// TwinCAT 3 PLC project machine1
// ProgramVersion: 3.1.4026.23
// CompilerDefines: VISU_USEPROPERTYINFO
// libraries:
//   CmpBitmapPool, * (System)
//   Tc2_Standard, * (Beckhoff Automation GmbH)
//   Tc2_System, * (Beckhoff Automation GmbH)
//   Tc2_Utilities, * (Beckhoff Automation GmbH)
//   Tc3_IotBase, * (Beckhoff Automation GmbH)
//   VisuDialogs, * (System)
// project tree:
//   DUTs/ E_SeqState.TcDUT
//   / GlobalTextList.TcGTLO, ImagePool.TcIPO (not stored), PlcTask.TcTTO, VisualizationManager.TcVMO (not stored)
//   GVLs/ GVL_IO.TcGVL, GVL_Nav.TcGVL, GVL_Param.TcGVL, GVL_Process.TcGVL, GVL_Secrets.TcGVL (not stored)
//   POUs/ FB_EventLog.TcPOU, MAIN.TcPOU, PRG_FileLogger.TcPOU, PRG_Params.TcPOU, PRG_Process.TcPOU, PRG_Spray.TcPOU, PRG_StatsLogger.TcPOU, PRG_Telegram.TcPOU, SIM_Plant.TcPOU
//   VISUs/ visu_Nav.TcVIS, visu_Params.TcVIS, visu_Spray.TcVIS
// real-time tasks:
//   TASK PlcTask: cycle T#10ms, priority 20, ADS port 350
// I/O:
//   DEVICE Device 1 (EtherCAT), AmsNetId 192.168.1.120.2.1
//     Term 1 (EK1100) [EK1100 EtherCAT Coupler (2A E-Bus)]
//       Term 2 (EL1859) [EL1859 8Ch. Dig. Input 24V, 3ms, 8Ch. Dig. Output 24V, 0.5A]
//       Term 3 (EL3054) [EL3054 4Ch. Ana. Input 4-20mA]
//       Term 4 (EL9011) [EL9011 End Terminal]
// variable links:
//   machine1/machine1 Instance <-> Device 1 (EtherCAT)/Term 1 (EK1100)/Term 2 (EL1859)
//     PlcTask Outputs/GVL_IO.bAirValve <-> Channel 9/Output
//   machine1/machine1 Instance <-> Device 1 (EtherCAT)/Term 1 (EK1100)/Term 3 (EL3054)
//     PlcTask Inputs/GVL_IO.iSPXLevelRaw <-> AI Standard Channel 1/Value

CONFIGURATION machine1
    RESOURCE PLC ON TwinCAT3
        TASK PlcTask(INTERVAL := T#10ms, PRIORITY := 20);
        PROGRAM MAIN WITH PlcTask : MAIN;
    END_RESOURCE
END_CONFIGURATION

// ---- DUTs/E_SeqState.TcDUT

{attribute 'strict'}
{attribute 'to_string'}
TYPE E_SeqState :
(
    eIdle         := 0,    // S0 - outputs safe, circulation on; wait for the mother handshake
    eDewater      := 10,   // S1 - T1 dewater (suck slurry); move mold to spray height
    eSprayOpen    := 20,   // S2 - open Air+SPX, piston OPENING; watchdogs T2 (valve) & T3 (piston)
    eSprayClose   := 30,   // S3 - piston CLOSING; watchdog T4; spraying continues
    eCloseDewater := 40,   // S4 - close Air+SPX (watchdog T6); T5 dewater; then release mother
    eFault        := 100   // FAULT - safe, latched until reset
) INT;
END_TYPE

// ---- GVLs/GVL_IO.TcGVL
// Physical process I/O, named per the Alfa/Brazil spec.
// Moved out of MAIN's VAR_INPUT/VAR_OUTPUT because several programs now
// touch these signals (MAIN sequence, PRG_Process supervision, PRG_Spray
// HMI, SIM_Plant). A GVL is the standard shared home - same reason the
// machine parameters already live in GVL_Param.
//
// For real hardware: replace ';' with the AT %I*/%Q* mappings noted on
// each line and set SIM_Plant.bSimEnable := FALSE.
{attribute 'qualified_only'}
VAR_GLOBAL
    // ============ DIGITAL INPUTS (0-24 V) ============
    // ---- SPX-valve traffic-light feedback ----
    bSPXFullyOpen    : BOOL;   // SPX valve reported FULLY OPEN     // AT %I*
    bSPXFullyClose   : BOOL;   // SPX valve reported FULLY CLOSED   // AT %I*
    // ---- piston position sensors (from the mother machine) ----
    bPistonClosed    : BOOL;   // 'P-close' - piston at closed end  // AT %I*
    bPistonOpen      : BOOL;   // 'P-open'  - piston at open end    // AT %I*
    // ---- mother-machine handshake ----
    bSprayFeasible   : BOOL;   // mother in position & waiting: we may run   // AT %I*
    bMoldAtSprayHigh : BOOL;   // 'spray height' - mold reached spray pos    // AT %I*
    // ---- operator pushbuttons (OR-ed with the HMI buttons in MAIN) ----
    bAutoToggleHW    : BOOL;   // HW AUTO/STOP toggle               // AT %I*
    bResetHW         : BOOL;   // HW fault reset                    // AT %I*

    // ============ ANALOG INPUTS (4-20 mA, scaled to engineering units) ============
	iSPXLevelRaw  AT %I* : INT; 
    rSPXLevel        : REAL;   // SPX tank level  [%]               // AT %I* (scaled)
    rSPXPressure     : REAL;   // SPX pressure    [bar]             // AT %I* (scaled)
    rAirPressure     : REAL;   // Air pressure    [bar]             // AT %I* (scaled)
    rPumpHzFb        : REAL;   // gear-pump ACTUAL speed [Hz]       // AT %I* (scaled)
                               // VFD speed feedback - the MEASURED counterpart of
                               // the rPumpHz setpoint below. The mimic (pump circle
                               // + Hz readout) shows this, never the command, so a
                               // dead drive cannot look like a running one.

    // ============ DIGITAL OUTPUTS (0-24 V) ============
    bAirValve  AT %Q*      : BOOL;   // air valve solenoid                // AT %Q*
    bSPXValve        : BOOL;   // SPX valve - command OPEN          // AT %Q*
    bCircValve       : BOOL;   // circulation valve = NOT bSPXValve // AT %Q*
    bPistonOpenSol   : BOOL;   // piston OPEN  solenoid (or mother cmd)  // AT %Q*
    bPistonCloseSol  : BOOL;   // piston CLOSE solenoid (or mother cmd)  // AT %Q*
    bGoToCleaningPos : BOOL;   // command mother: move mold to spray height  // AT %Q*
    bSprayBusy       : BOOL;   // handshake to mother: we are running (mother waits)  // AT %Q*

    // ============ ANALOG OUTPUT (4-20 mA) ============
    rPumpHz          : REAL;   // gear-pump VFD speed setpoint [Hz] // AT %Q* (scaled)
END_VAR

// ---- GVLs/GVL_Nav.TcGVL
// Navigation state shared by the screen programs.
// Two screens now, per the spec.
{attribute 'qualified_only'}
VAR_GLOBAL
    nPage       : INT;                   // 0 = Spray System, 1 = Machine Parameters
    abNavActive : ARRAY[0..1] OF BOOL;   // highlight for the active nav button
END_VAR

// ---- GVLs/GVL_Param.TcGVL
// Machine parameters - persistent, writable from PRG_Params, read everywhere.
// Defaults match the "Machine Parameters" screen in the spec.
//   *** marks values the spec left open ("??"/"X"); tune on the machine. ***
{attribute 'qualified_only'}
VAR_GLOBAL PERSISTENT
    // ===== sequence timers (HMI "Machine Parameters" page) =====
    tDewaterTime       : TIME := T#4S;     // T1 - dewater / suck slurry            [operator]
    tSPXMaxOpenTime    : TIME := T#500MS;  // T2 - SPX valve must report OPEN  within this  [engineer]
    tSPXMaxCloseTime   : TIME := T#500MS;  // T6 - SPX valve must report CLOSE within this  [engineer]  (HMI groups T2&T6)
    tSprayOpenTime     : TIME := T#3S;     // T3 - piston OPEN  stroke watchdog (P-close->P-open) [engineer]
    tSprayCloseTime    : TIME := T#3S;     // T4 - piston CLOSE stroke watchdog (P-open->P-close) [engineer]  (HMI groups T3&T4)
    tSPXDewaterTime    : TIME := T#10S;    // T5 - dewater after closing            [operator]

    // ===== pressure / pump (HMI "Machine Parameters" page) =====
    rSPXPressureTarget : REAL := 1.7;      // SPX target pressure [bar]
    rPumpSpeedBase     : REAL := 15.0;     // gear-pump base speed [Hz] (P-control starts here)

    // ===== thresholds & gains (engineer; not on the operator page) =====
    rSPXPressTol       : REAL := 0.1;      // |avg-target| >= this  -> "bad SPX pressure" warning
    rPumpDeadband      : REAL := 0.02;     // P-control deadband [bar]
    rPumpKp            : REAL := 2.0;      // *** P-control gain [Hz per bar] - spec: "double the difference??" ***
    rPumpHzMin         : REAL := 5.0;      // *** pump speed clamp, low  [Hz] ***
    rPumpHzMax         : REAL := 50.0;     // *** pump speed clamp, high [Hz] ***
    rLevelHigh         : REAL := 95.0;     // SPX tank: warn above [%]
    rLevelLow          : REAL := 20.0;     // SPX tank: warn below [%]
    rLevelEmpty        : REAL := 5.0;      // SPX tank: below -> stop pump & block mother release [%]
    rCircPressTol      : REAL := 0.5;      // spray-avg vs circulation-avg > this -> "adjust" message

    // ===== logging =====
    // Directory for the event log file (PRG_FileLogger).
    //   ''  -> TwinCAT boot folder of the TARGET (portable default:
    //          Windows C:\TwinCAT\3.1\Boot\ , BSD/Linux /usr/local/etc/TwinCAT/3.1/Boot/)
    //   'C:\kayma\machine1'          -> Windows dev PC
    //   '/home/Administrator/logs'   -> Linux/BSD PLC (folder must exist & be writable
    //                                   by the TwinCAT runtime user!)
    // PERSISTENT: set once per machine, survives reboots. Takes effect on the
    // next logged event - no restart needed.
    sLogDir            : STRING(255) := '';

    // TRUE  -> every sequence state transition is logged as INFO
    //          (~4 extra lines per spray cycle; great for commissioning)
    // FALSE -> only cycle start/complete, faults, resets, warnings
    bLogStateChanges   : BOOL := TRUE;
	bStatsEnable   : BOOL := TRUE;   // master switch
    tStatsRun      : TIME := T#1S;   // sample period while cycle active
    tStatsIdle     : TIME := T#2M;   // keep-alive period idle/fault
    nStatsHourFrom : INT  := 0;      // daily window; From=To=0 -> 24h
    nStatsHourTo   : INT  := 0;      // e.g. 6 & 22 -> log 06:00-21:59
END_VAR

VAR_GLOBAL CONSTANT
    // ===== factory defaults (RESET button on the params page) =====
    // One authoritative home for the default machine parameters.
    // If you retune the machine, change the defaults HERE (they should
    // normally mirror the init values of the persistent block above).
    cDefDewaterTime    : TIME := T#4S;      // T1
    cDefValveMaxTime   : TIME := T#500MS;   // T2 & T6
    cDefSprayTime      : TIME := T#3S;      // T3 & T4
    cDefSPXDewaterTime : TIME := T#10S;     // T5
    cDefPressTarget    : REAL := 1.7;       // [bar]
    cDefPumpSpeed      : REAL := 15.0;      // [Hz]
END_VAR

// ---- GVLs/GVL_Process.TcGVL
// Derived process values + non-latching warnings.
//   - MAIN accumulates the SPX pressure averages during T3/T4.
//   - PRG_Process uses them for the end-of-cycle pump correction and
//     computes the level/circulation warnings.
//   - PRG_Spray shows them.
// (Sequence FAULTS are separate and latched - see MAIN.nErrorCode.)
{attribute 'qualified_only'}
VAR_GLOBAL
    // ---- SPX pressure averaging ----
    rSPXAvgT3      : REAL;   // "SPX Pressure average at T3"  (opening stroke)
    rSPXAvgT4      : REAL;   // "SPX Pressure average at T4"  (closing stroke)
    rSPXAvg        : REAL;   // "SPX Pressure average" = mean(T3, T4); drives pump P-control
    rSPXAvgCirc    : REAL;   // SPX pressure average during circulation (handshake down)

    // ---- warnings (non-latching; shown on the Spray screen) ----
    bWarnBadSPX    : BOOL;   // |spray avg - target| >= rSPXPressTol  ("bad SPX pressure")
    bWarnLevelHigh : BOOL;   // level > rLevelHigh
    bWarnLevelLow  : BOOL;   // level < rLevelLow
    bLevelEmpty    : BOOL;   // level < rLevelEmpty -> pump off + mother release blocked
    bWarnCircPress : BOOL;   // spray avg differs from circulation avg by > rCircPressTol ("adjust")
END_VAR

// ---- POUs/MAIN.TcPOU
PROGRAM MAIN
VAR_OUTPUT
    // ---- status (read by the HMI screens) ----
    eState        : E_SeqState := E_SeqState.eIdle;  // current sequence state
    nErrorCode    : INT;          // latched sequence fault (see constants)
    bAutoMode     : BOOL;         // TRUE = AUTO armed.  FALSE at boot = MANUAL
    bError        : BOOL;         // TRUE while in fault
    bReadyToStart : BOOL;         // TRUE while idle in manual (AUTO can be armed)
END_VAR

VAR
    // ---- edge detection ----
    rtAuto  : R_TRIG;   // AUTO/STOP toggle (HW OR HMI)
    rtReset : R_TRIG;   // fault reset      (HW OR HMI)

    // ---- timers (one per spec timer) ----
    tonDewater    : TON;   // T1 - dewater / suck slurry
    tonSPXOpen    : TON;   // T2 - SPX-valve-open watchdog
    tonSprayOpen  : TON;   // T3 - piston opening-stroke watchdog
    tonSprayClose : TON;   // T4 - piston closing-stroke watchdog
    tonSPXClose   : TON;   // T6 - SPX-valve-close watchdog
    tonDewaterCl  : TON;   // T5 - dewater after closing

    // ---- SPX pressure averaging accumulators ----
    rSumT3   : REAL;   nCntT3   : DINT;   // opening stroke
    rSumT4   : REAL;   nCntT4   : DINT;   // closing stroke
    rSumCirc : REAL;   nCntCirc : DINT;   // circulation (handshake down)
END_VAR

VAR CONSTANT
    // ---- latched fault codes ----
    nERR_NONE            : INT := 0;
    nERR_PISTON_NOT_HOME : INT := 10;   // start: piston not at P-close
    nERR_SPX_OPEN_STUCK  : INT := 20;   // T2: SPX valve never reported Fully Open
    nERR_SPX_CLOSE_STUCK : INT := 21;   // T6: SPX valve never reported Fully Close
    nERR_PISTON_OPEN_TO  : INT := 30;   // T3: piston did not reach P-open in time
    nERR_PISTON_CLOSE_TO : INT := 40;   // T4: piston did not reach P-close in time
	nERR_LEVEL_HIGH : INT := 50;   // SPX level above rLevelHigh (>95%)
	nERR_LEVEL_LOW  : INT := 51;   // SPX level below rLevelEmpty (<5%)
    nERR_UNKNOWN_STATE   : INT := 99;   // illegal eState

    // level fault auto-clear hysteresis [%]: the level must come back
    // this far INSIDE the band before the fault self-clears, so the
    // fault cannot chatter on/off right at the threshold.
    rLEVEL_CLEAR_HYST    : REAL := 2.0;
END_VAR

//==================================================================
// MAIN - spray sequence + scheduling   (aligned to the Alfa/Brazil spec)
//
// Flow (AUTO):  mother raises 'Spray feasible' -> we take control, move
// the mold to spray height, run ONE spray cycle (T1..T6), then lower
// 'busy' so the mother resumes. The cycle is handshake-gated, not free-
// running: each casting cycle the mother hands us control exactly once.
//==================================================================
SIM_Plant();    // drives GVL_IO inputs; bSimEnable is the sim/real master (HMI button)

// Scale EL3054 raw (0..32767 = 4..20 mA) -> SPX tank level [%].
// Only with REAL VALUES selected: while simulating, SIM_Plant ramps
// rSPXLevel and this must not overwrite it. Same single flag that
// gates every other input, so the level can never end up on a
// different source than the rest of the screen.
IF NOT SIM_Plant.bSimEnable THEN
    GVL_IO.rSPXLevel := INT_TO_REAL(GVL_IO.iSPXLevelRaw) * (100.0 / 32767.0);
END_IF

// Edge detectors (HW inputs OR-ed with the HMI buttons from PRG_Spray).
rtAuto (CLK := GVL_IO.bAutoToggleHW OR PRG_Spray.bCmdAuto);
rtReset(CLK := GVL_IO.bResetHW      OR PRG_Spray.bCmdReset);

// The circulation valve is ALWAYS the inverse of the SPX valve.
GVL_IO.bCircValve := NOT GVL_IO.bSPXValve;

// ---- AUTO / MANUAL toggle ----
//   press once  -> arm AUTO
//   AUTO -> MANUAL -> STOP NOW: abort to S0/idle on THIS scan. Because
//   this runs before the CASE, the eIdle branch below drops every
//   actuator the same scan - the running cycle stops immediately.
IF rtAuto.Q THEN
    IF bAutoMode THEN
        bAutoMode := FALSE;                 // AUTO -> MANUAL
        eState    := E_SeqState.eIdle;      // abort to S0 immediately (outputs drop in eIdle)
    ELSIF NOT bError THEN
        bAutoMode := TRUE;                  // arm AUTO
    END_IF
END_IF

CASE eState OF

    //--------------------------------------------------------------
    // S0 - IDLE / MANUAL   (circulation running, mother free)
    //--------------------------------------------------------------
    E_SeqState.eIdle:
        GVL_IO.bAirValve        := FALSE;
        GVL_IO.bSPXValve        := FALSE;     // -> circulation valve open
        GVL_IO.bPistonCloseSol  := TRUE;      // default: hold the piston closed
        GVL_IO.bPistonOpenSol   := FALSE;
        GVL_IO.bGoToCleaningPos := FALSE;
        GVL_IO.bSprayBusy       := FALSE;     // mother is free to move
        bError        := FALSE;
        bReadyToStart := NOT bAutoMode;
        nErrorCode    := nERR_NONE;

        // reset all timers + stroke accumulators (clean start next cycle)
        tonDewater(IN := FALSE);   tonSPXOpen(IN := FALSE);   tonSprayOpen(IN := FALSE);
        tonSprayClose(IN := FALSE); tonSPXClose(IN := FALSE); tonDewaterCl(IN := FALSE);
        rSumT3 := 0; nCntT3 := 0; rSumT4 := 0; nCntT4 := 0;

        // average SPX pressure during circulation (handshake down)
        rSumCirc := rSumCirc + GVL_IO.rSPXPressure;
        nCntCirc := nCntCirc + 1;
        IF nCntCirc > 0 THEN
            GVL_Process.rSPXAvgCirc := rSumCirc / DINT_TO_REAL(nCntCirc);
        END_IF

        IF bAutoMode THEN
            // Start a cycle only when the mother hands control over
            // (bSprayFeasible), the piston is home, and the tank isn't empty.
            IF GVL_IO.bSprayFeasible AND GVL_IO.bPistonClosed AND NOT GVL_Process.bLevelEmpty THEN
                GVL_IO.bSprayBusy       := TRUE;   // tell the mother we are running
                GVL_IO.bGoToCleaningPos := TRUE;   // ask the mother to move the mold up
                GVL_Process.bWarnBadSPX := FALSE;  // fresh cycle
                rSumCirc := 0; nCntCirc := 0;      // restart circulation average
                bReadyToStart := FALSE;
                eState := E_SeqState.eDewater;
            END_IF
        ELSIF PRG_Spray.bManualActive THEN
            // MANUAL: operator drives the actuators directly.
            GVL_IO.bAirValve       := PRG_Spray.bManAirValve;
            GVL_IO.bSPXValve       := PRG_Spray.bManSPXValve;
            GVL_IO.bPistonOpenSol  := PRG_Spray.bManPistonOpen;
            GVL_IO.bPistonCloseSol := PRG_Spray.bManPistonClose;
        END_IF

    //--------------------------------------------------------------
    // S1 - DEWATER (T1)   + position the mold to spray height
    //--------------------------------------------------------------
    E_SeqState.eDewater:
        GVL_IO.bAirValve       := FALSE;
        GVL_IO.bSPXValve       := FALSE;
        GVL_IO.bPistonCloseSol := TRUE;       // keep piston closed
        GVL_IO.bPistonOpenSol  := FALSE;

        // keep asking until the mold reports it is at spray height
        GVL_IO.bGoToCleaningPos := NOT GVL_IO.bMoldAtSprayHigh;

        tonDewater(IN := TRUE, PT := GVL_Param.tDewaterTime);

        // advance once T1 elapsed AND the mold is in position
        IF tonDewater.Q AND GVL_IO.bMoldAtSprayHigh THEN
            eState := E_SeqState.eSprayOpen;
        END_IF

    //--------------------------------------------------------------
    // S2 - SPRAY, OPENING   (open valves; piston travels P-close->P-open)
    //   T2 watchdog: SPX valve must reach Fully Open.
    //   T3 watchdog: piston must complete the opening stroke.
    //   Average SPX pressure over the stroke -> "...average at T3".
    //--------------------------------------------------------------
    E_SeqState.eSprayOpen:
        GVL_IO.bAirValve       := TRUE;
        GVL_IO.bSPXValve       := TRUE;       // -> circulation valve closes
        GVL_IO.bPistonOpenSol  := TRUE;       // drive piston OPEN
        GVL_IO.bPistonCloseSol := FALSE;

        // T2 - SPX-valve-open confirmation watchdog (runs until Fully Open)
        tonSPXOpen(IN := NOT GVL_IO.bSPXFullyOpen, PT := GVL_Param.tSPXMaxOpenTime);
        IF tonSPXOpen.Q THEN
            nErrorCode := nERR_SPX_OPEN_STUCK;
            eState     := E_SeqState.eFault;
        END_IF

        // T3 - opening-stroke watchdog (starts once the piston leaves P-close)
        tonSprayOpen(IN := NOT GVL_IO.bPistonClosed, PT := GVL_Param.tSprayOpenTime);
        IF tonSprayOpen.Q AND NOT GVL_IO.bPistonOpen THEN
            nErrorCode := nERR_PISTON_OPEN_TO;
            eState     := E_SeqState.eFault;
        END_IF

        // running SPX pressure average over the opening stroke
        rSumT3 := rSumT3 + GVL_IO.rSPXPressure;
        nCntT3 := nCntT3 + 1;

        // stroke finished -> store average, check pressure, go to closing
        IF GVL_IO.bPistonOpen THEN
            IF nCntT3 > 0 THEN
                GVL_Process.rSPXAvgT3 := rSumT3 / DINT_TO_REAL(nCntT3);
            END_IF
            IF ABS(GVL_Process.rSPXAvgT3 - GVL_Param.rSPXPressureTarget) >= GVL_Param.rSPXPressTol THEN
                GVL_Process.bWarnBadSPX := TRUE;
            END_IF
            eState := E_SeqState.eSprayClose;
        END_IF

    //--------------------------------------------------------------
    // S3 - SPRAY, CLOSING   (piston travels P-open->P-close)
    //   T4 watchdog: piston must complete the closing stroke.
    //   Average SPX pressure over the stroke -> "...average at T4".
    //--------------------------------------------------------------
    E_SeqState.eSprayClose:
        GVL_IO.bAirValve       := TRUE;
        GVL_IO.bSPXValve       := TRUE;
        GVL_IO.bPistonOpenSol  := FALSE;
        GVL_IO.bPistonCloseSol := TRUE;       // drive piston CLOSE

        // T4 - closing-stroke watchdog (starts once the piston leaves P-open)
        tonSprayClose(IN := NOT GVL_IO.bPistonOpen, PT := GVL_Param.tSprayCloseTime);
        IF tonSprayClose.Q AND NOT GVL_IO.bPistonClosed THEN
            nErrorCode := nERR_PISTON_CLOSE_TO;
            eState     := E_SeqState.eFault;
        END_IF

        rSumT4 := rSumT4 + GVL_IO.rSPXPressure;
        nCntT4 := nCntT4 + 1;

        IF GVL_IO.bPistonClosed THEN
            IF nCntT4 > 0 THEN
                GVL_Process.rSPXAvgT4 := rSumT4 / DINT_TO_REAL(nCntT4);
            END_IF
            IF ABS(GVL_Process.rSPXAvgT4 - GVL_Param.rSPXPressureTarget) >= GVL_Param.rSPXPressTol THEN
                GVL_Process.bWarnBadSPX := TRUE;
            END_IF
            eState := E_SeqState.eCloseDewater;
        END_IF

    //--------------------------------------------------------------
    // S4 - CLOSE + DEWATER   (T6 valve-close watchdog + T5 dewater)
    //   On T5 end: lower 'busy' -> the mother resumes.
    //--------------------------------------------------------------
    E_SeqState.eCloseDewater:
        GVL_IO.bAirValve       := FALSE;
        GVL_IO.bSPXValve       := FALSE;      // -> circulation valve opens again
        GVL_IO.bPistonOpenSol  := FALSE;
        GVL_IO.bPistonCloseSol := TRUE;       // hold piston closed

        // T6 - SPX-valve-close confirmation watchdog (runs until Fully Close)
        tonSPXClose(IN := NOT GVL_IO.bSPXFullyClose, PT := GVL_Param.tSPXMaxCloseTime);
        IF tonSPXClose.Q THEN
            nErrorCode := nERR_SPX_CLOSE_STUCK;
            eState     := E_SeqState.eFault;
        END_IF

        // T5 - dewater
        tonDewaterCl(IN := TRUE, PT := GVL_Param.tSPXDewaterTime);
        IF tonDewaterCl.Q THEN
            // tank-empty lockout: do NOT release the mother while empty
            IF NOT GVL_Process.bLevelEmpty THEN
                GVL_IO.bSprayBusy := FALSE;          // lower the flag -> mother resumes
                eState            := E_SeqState.eIdle;
            END_IF
        END_IF

    //--------------------------------------------------------------
    // FAULT - latched until reset.
    //   The actuators are forced safe by the SAFE-STATE OVERLAY right
    //   after this CASE, so a fault raised mid-cycle drops every output
    //   on the SAME scan (the spray states energise their outputs at the
    //   top of their branch, then test for faults).
    //--------------------------------------------------------------
    E_SeqState.eFault:
        // LEVEL faults (50/51) self-clear as soon as the operator brings
        // the tank back into band (refill after "low", drain after "high"),
        // with hysteresis so the fault can't chatter at the threshold.
        // Every other fault stays latched until Reset.
        // NOTE: the safe-state overlay already dropped AUTO -> MANUAL, so
        // after the auto-clear the machine sits safely in Idle/MANUAL and
        // the operator re-arms AUTO deliberately.
        IF rtReset.Q
        OR (nErrorCode = nERR_LEVEL_LOW  AND GVL_IO.rSPXLevel >= GVL_Param.rLevelEmpty + rLEVEL_CLEAR_HYST)
        OR (nErrorCode = nERR_LEVEL_HIGH AND GVL_IO.rSPXLevel <= GVL_Param.rLevelHigh  - rLEVEL_CLEAR_HYST) THEN
            bError     := FALSE;
            nErrorCode := nERR_NONE;
            eState     := E_SeqState.eIdle;
        END_IF

ELSE
    nErrorCode := nERR_UNKNOWN_STATE;
    eState     := E_SeqState.eFault;
END_CASE

//==================================================================
// SPX LEVEL FAULT - out-of-band level raises a latched fault,
//   but ONLY while AUTO is armed or a spray cycle is running.
//   >95% = overfill,  <5% = dry/disconnected.
//   In MANUAL + idle (operator draining / refilling / cleaning) NO
//   fault is raised - the machine is still protected by:
//     - the non-latching warnings on the Spray screen (PRG_Process)
//     - the tank-empty pump lockout in PRG_Process (pump -> 0 Hz)
//     - the AUTO start gate in eIdle (NOT bLevelEmpty)
//   The fault self-clears in eFault once the level is back in band
//   (see the eFault branch above); Reset also still works.
//==================================================================
IF eState <> E_SeqState.eFault AND (bAutoMode OR eState <> E_SeqState.eIdle) THEN
    IF GVL_IO.rSPXLevel > GVL_Param.rLevelHigh THEN
        nErrorCode := nERR_LEVEL_HIGH;
        eState     := E_SeqState.eFault;
    ELSIF GVL_IO.rSPXLevel < GVL_Param.rLevelEmpty THEN
        nErrorCode := nERR_LEVEL_LOW;
        eState     := E_SeqState.eFault;
    END_IF
END_IF

//==================================================================
// SAFE-STATE OVERLAY - runs every scan, right after the sequencer.
//   A fault must stop the process RIGHT AWAY. The spray states set
//   their outputs TRUE at the top of the branch and only then test for
//   faults, so without this the actuators would drop one scan late. On
//   the scan a fault is raised, eState is already eFault here, so every
//   output drops in the same scan and AUTO is dropped to MANUAL.
//   (The AUTO->MANUAL abort lands in eIdle above, which is safe the
//    same scan, so it needs no overlay.)
//==================================================================
IF eState = E_SeqState.eFault THEN
    GVL_IO.bAirValve        := FALSE;
    GVL_IO.bSPXValve        := FALSE;
    GVL_IO.bPistonOpenSol   := FALSE;
    GVL_IO.bPistonCloseSol  := TRUE;     // hold the piston closed
    GVL_IO.bGoToCleaningPos := FALSE;
    GVL_IO.bSprayBusy       := FALSE;    // hand control back to the mother
    bError        := TRUE;
    bReadyToStart := FALSE;
    bAutoMode     := FALSE;              // a fault always drops AUTO -> MANUAL
END_IF

//==================================================================
// Supervision + screen programs (all run every scan)
//==================================================================
PRG_Process();   // level monitoring, pump P-control, circulation check
PRG_Spray();     // Spray System screen      (page 0)
PRG_Params();    // Machine Parameters screen (page 1)
PRG_FileLogger(); // Logger for the machine
PRG_Telegram();  // Telegram fault notifier (TF6760)

END_PROGRAM

// ---- POUs/SIM_Plant.TcPOU
PROGRAM SIM_Plant
//==================================================================
// PLANT SIMULATOR - drives the GVL_IO *inputs* from the GVL_IO outputs
// so the aligned sequence can run without hardware. Stroke/valve times
// are set INSIDE the watchdog limits (T2/T3/T4/T6) so a clean demo
// never faults. Set bSimEnable := FALSE for real I/O.
//
// bSimEnable is the ONE switch: it is what the 'SIM VALUES / REAL
// VALUES' button on the spray screen toggles, and it covers every
// process input at once (level, pressures, pump speed feedback, valve
// traffic-light, piston sensors, mold-at-height, mother handshake).
// On the falling
// edge the simulated values are dropped rather than left latched -
// see the release block at the top of the implementation.
//==================================================================
VAR
    bSimEnable       : BOOL := TRUE;     // master enable (HMI: 'SIM VALUES' button)
    bSimAutoStart    : BOOL := FALSE;    // TRUE = kick the machine into AUTO once (demo).
                                         // Default FALSE: boots in MANUAL, as specified.
	ftSimOff        : F_TRIG;         // SIM -> REAL edge (release the sim values)
    fSimLevel       : REAL := 20.0;   // simulated level [%]
    fSimRate        : REAL := 5.0;    // rate of change [% per second]
    bSimUp          : BOOL := TRUE;   // TRUE = filling, FALSE = draining
	bAutoKicked 	: BOOL;
    tLast           : TIME;
    fDt             : REAL;

    // ---- simulated mechanical times (must stay < the matching watchdog) ----
    tSimPistonStroke : TIME := T#2S;     // piston travel  (< T3 / T4 = 3 s)
    tSimValveStroke  : TIME := T#300MS;  // SPX valve open/close (< T2 / T6 = 0.5 s)
    tSimMoldMove     : TIME := T#1S;     // mother moves mold to spray height (< T1 = 4 s)
    tSimStartGap     : TIME := T#2S;     // settle time before the demo auto-kick

    // ---- simulated VFD speed feedback ----
    rSimPumpLag      : REAL := 0.15;  // per-scan approach factor -> spin-up/down
    rSimPumpZero     : REAL := 0.5;   // [Hz] snap the lag tail to 0 below this.
                                      // Keep at/below PRG_Spray.rPUMP_RUN_MIN, the
                                      // threshold the mimic calls 'stopped'.

    // ---- timers ----
    tonPOpen   : TON;
    tonPClose  : TON;
    tonSPXO    : TON;
    tonSPXC    : TON;
    tonMold    : TON;
    tonStart   : TON;
    rtStartGap : R_TRIG;
    
END_VAR

//------------------------------------------------------------------
// Simulation off -> leave every input to the real I/O.
//   On the SIM -> REAL edge the values this program was writing are
//   cleared. Without that they stay latched at their last simulated
//   figure and keep reading like live measurements - the piston lamps
//   stay green, SPX still shows 1.72 bar - which is exactly the trap
//   the sim/real button exists to prevent. Zeroed inputs make an
//   unmapped or dead channel obvious immediately (and, in AUTO, the
//   existing watchdogs fault the cycle instead of running blind).
//------------------------------------------------------------------
ftSimOff(CLK := bSimEnable);

IF NOT bSimEnable THEN
    IF ftSimOff.Q THEN
        GVL_IO.rSPXPressure     := 0.0;
        GVL_IO.rAirPressure     := 0.0;
        GVL_IO.rPumpHzFb        := 0.0;
        GVL_IO.bSPXFullyOpen    := FALSE;
        GVL_IO.bSPXFullyClose   := FALSE;
        GVL_IO.bPistonOpen      := FALSE;
        GVL_IO.bPistonClosed    := FALSE;
        GVL_IO.bMoldAtSprayHigh := FALSE;
        GVL_IO.bSprayFeasible   := FALSE;
        GVL_IO.bAutoToggleHW    := FALSE;
        // rSPXLevel is not cleared here: MAIN scales it from the real
        // iSPXLevelRaw channel every scan as soon as sim is off.
    END_IF
    RETURN;
END_IF

//------------------------------------------------------------------
// Mother handshake: mother is always ready in the demo, so each time
// the cycle returns to idle it hands control over again (cycles loop).
//------------------------------------------------------------------
GVL_IO.bSprayFeasible := TRUE;

//------------------------------------------------------------------
// Piston position sensors (P-close / P-open) follow the solenoids.
//   leaving an end clears that end immediately; reaching the far end
//   takes tSimPistonStroke.
//------------------------------------------------------------------
tonPOpen (IN := GVL_IO.bPistonOpenSol,  PT := tSimPistonStroke);
tonPClose(IN := GVL_IO.bPistonCloseSol, PT := tSimPistonStroke);

IF GVL_IO.bPistonOpenSol THEN
    GVL_IO.bPistonClosed := FALSE;
    GVL_IO.bPistonOpen   := tonPOpen.Q;
ELSIF GVL_IO.bPistonCloseSol THEN
    GVL_IO.bPistonOpen   := FALSE;
    GVL_IO.bPistonClosed := tonPClose.Q;
END_IF

//------------------------------------------------------------------
// SPX valve traffic-light follows the SPX valve command.
//------------------------------------------------------------------
tonSPXO(IN := GVL_IO.bSPXValve,     PT := tSimValveStroke);
tonSPXC(IN := NOT GVL_IO.bSPXValve, PT := tSimValveStroke);

IF GVL_IO.bSPXValve THEN
    GVL_IO.bSPXFullyClose := FALSE;
    GVL_IO.bSPXFullyOpen  := tonSPXO.Q;
ELSE
    GVL_IO.bSPXFullyOpen  := FALSE;
    GVL_IO.bSPXFullyClose := tonSPXC.Q;
END_IF

//------------------------------------------------------------------
// Mold reaches spray height shortly after we take control (busy).
//------------------------------------------------------------------
tonMold(IN := GVL_IO.bSprayBusy, PT := tSimMoldMove);
GVL_IO.bMoldAtSprayHigh := tonMold.Q;

//------------------------------------------------------------------
// Analog inputs.  Level mid-range (no level warnings); SPX pressure
// eases toward ~1.72 bar while spraying (within tolerance of 1.70).
//------------------------------------------------------------------

IF GVL_IO.bSPXValve THEN
    GVL_IO.rSPXPressure := GVL_IO.rSPXPressure + (1.72 - GVL_IO.rSPXPressure) * 0.3;
ELSE
    GVL_IO.rSPXPressure := GVL_IO.rSPXPressure + (1.50 - GVL_IO.rSPXPressure) * 0.1;
END_IF

IF GVL_IO.bAirValve THEN
    GVL_IO.rAirPressure := GVL_IO.rAirPressure + (28.0 - GVL_IO.rAirPressure) * 0.3;
ELSE
    GVL_IO.rAirPressure := GVL_IO.rAirPressure + (5.0 - GVL_IO.rAirPressure) * 0.1;
END_IF

//------------------------------------------------------------------
// Gear-pump speed feedback: first-order lag toward the VFD setpoint,
// i.e. spin-up and spin-down instead of an instant jump. The setpoint
// read here is the one written LAST scan (PRG_Process / PRG_Spray both
// run after this program), which is the right way round - a real drive
// reports where it has got to, not where it was just told to go.
// Snapped to exactly 0 below the run threshold: the lag is asymptotic,
// and a stopped pump must read zero rather than leave a tail that
// keeps the mimic circle green forever.
//------------------------------------------------------------------
GVL_IO.rPumpHzFb := GVL_IO.rPumpHzFb + (GVL_IO.rPumpHz - GVL_IO.rPumpHzFb) * rSimPumpLag;
IF GVL_IO.rPumpHz <= 0.0 AND GVL_IO.rPumpHzFb < rSimPumpZero THEN
    GVL_IO.rPumpHzFb := 0.0;
END_IF

//------------------------------------------------------------------
// Demo kick-off: pulse the AUTO toggle ONCE after boot (if enabled).
// Cycles then loop on their own (machine stays armed in AUTO), so we
// must NOT pulse again - a second pulse would disarm AUTO.
//------------------------------------------------------------------
tonStart(IN := bSimAutoStart AND NOT bAutoKicked AND (MAIN.eState = E_SeqState.eIdle),
         PT := tSimStartGap);
rtStartGap(CLK := tonStart.Q);
GVL_IO.bAutoToggleHW := rtStartGap.Q;
IF rtStartGap.Q THEN
    bAutoKicked := TRUE;
END_IF

fDt   := TIME_TO_REAL(TIME() - tLast) / 1000.0;
tLast := TIME();
fDt   := LIMIT(0.0, fDt, 0.1);   // guard against the first-cycle jump

// Level ramp - unconditional while simulating, like every other value
// this program drives. (There used to be a bSimLevelActive sub-flag
// that could hold the level on the real channel while the rest of the
// screen was simulated; with bSimEnable on the HMI it was a second,
// unreachable switch that silently froze the level. One switch only.)
IF bSimUp THEN
    fSimLevel := fSimLevel + fSimRate * fDt;
    IF fSimLevel >= 90.0 THEN
        fSimLevel := 90.0;
        bSimUp    := FALSE;      // top reached -> drain
    END_IF
ELSE
    fSimLevel := fSimLevel - fSimRate * fDt;
    IF fSimLevel <= 21.0 THEN
        fSimLevel := 21.0;
        bSimUp    := TRUE;       // bottom reached -> fill
    END_IF
END_IF
GVL_IO.rSPXLevel := fSimLevel;

END_PROGRAM

// ---- POUs/PRG_Spray.TcPOU
PROGRAM PRG_Spray
//==================================================================
// SPRAY SYSTEM SCREEN  (page 0)
//   The mimic view from the spec (slide 12). Merges the three old
//   spray programs (process view + manual + live readouts) into one
//   schematic screen:
//     - valve states by colour: green = open, grey = closed,
//       red = in transit (SPX by traffic-light, circulation = inverse,
//       air by command)
//     - piston lamps (green at a known end), mold-at-height lamp,
//       spray marks, pump Hz, SPX level, SPX/Air pressures
//     - manual buttons (live only in manual); mode colour
//       yellow = manual, green = auto
//     - CLEAN MODE (manual only): drain tank -> close drain / add
//       water prompts -> refill to 20% -> 20 s delay -> auto-open
//       the SPX valve to flush the pipes (section 6b)
//   The sequence engine stays in MAIN; this program is the HMI face.
//==================================================================
VAR_OUTPUT
    // ---- operator commands consumed by MAIN ----
    bCmdAuto  : BOOL;    // AUTO/MANUAL toggle button (tap = pulse)
    bCmdReset : BOOL;    // "Reset fault" button

    // ---- manual mode (consumed by MAIN while idle) ----
    bManualActive   : BOOL;   // TRUE = manual commands drive the outputs
    bManAirValve    : BOOL;   // manual: air valve        (HMI toggle)
    bManSPXValve    : BOOL;   // manual: SPX valve         (HMI toggle)
    bManPistonOpen  : BOOL;   // manual: piston OPEN  sol. (HMI toggle)
    bManPistonClose : BOOL;   // manual: piston CLOSE sol. (HMI toggle)
    rManPumpHz      : REAL := 15.0;   // manual/clean pump speed [Hz] - mirrors GVL_Param.rPumpSpeedBase every scan

    // ---- clean mode (read by MAIN) ----
    bCleanActive    : BOOL;   // TRUE = clean sequence running: MAIN skips the
                              // level-LOW fault and refuses to arm AUTO
    bPostCleanEmpty : BOOL;   // TRUE = clean ended with a dry tank: keep the
                              // level-LOW fault suppressed until refilled >5%
END_VAR

VAR
	
 	// ---- readout text colours (AARRGGBB) ----
    //   black = normal, amber = warning, red = lockout. Driven from the flags
    //   PRG_Process/MAIN already evaluate, so the colour on screen can never
    //   disagree with the fault code or the log file.
    cSPXPress   : DWORD;   // SPX pressure field. Amber while GVL_Process.bWarnBadSPX,
                           // i.e. the last cycle's T3/T4 average sat further than
                           // rSPXPressTol from rSPXPressureTarget. Latched per cycle,
                           // so it describes the last spray, not the live number.
    cLevel      : DWORD;   // SPX level field. Amber below rLevelLow or above
                           // rLevelHigh, red below rLevelEmpty (bLevelEmpty, which
                           // also stops the pump and blocks the mother release).
    // ---- mimic colours (AARRGGBB) ----
    cAirValve   : DWORD;
    cSPXValve   : DWORD;
    cCircValve  : DWORD;
    cPistonOpen : DWORD;
    cPistonClose: DWORD;
    cModeColor  : DWORD;

    // ---- lamps / flags ----
    bMoldLamp   : BOOL;   // mold at spray height
    bSprayMarks : BOOL;   // spray marks visible
    bFault      : BOOL;

    // ---- text ----
    sStateText  : STRING;
    sModeText   : STRING;
    sErrorText  : STRING;
    sWarnText   : STRING;

    // ---- live readouts mirrored for the HMI ----
    rPumpHz      : REAL;
    rSPXLevel    : REAL;
    rSPXPressure : REAL;
    rAirPressure : REAL;

    // ---- clean mode: HMI buttons (Toggle inputs; consumed in section 7) ----
    bBtnClean      : BOOL;   // 'CLEAN MODE' / 'STOP CLEAN' button
    bBtnStartClean : BOOL;   // 'Start Clean' button
    bBtnCloseDrain : BOOL;   // 'Close Drain' acknowledge button
    bBtnAddWater   : BOOL;   // 'Add Water'  acknowledge button

    // ---- clean mode: state + HMI feedback ----
    nCleanStep     : INT;    // nCLEAN_* constants below
    bDrainAck      : BOOL;   // operator confirmed the drain is closed
    bWaterAck      : BOOL;   // operator confirmed water is being added
    bDrainFlash    : BOOL;   // bind to 'Close Drain' toggle-colour -> flashes
    bWaterFlash    : BOOL;   // bind to 'Add Water'  toggle-colour -> flashes
    sCleanBtnText  : STRING := 'CLEAN MODE';  // 'CLEAN MODE' <-> 'STOP CLEAN'
    sCleanStatus   : STRING; // one-line operator guidance + countdown
    nFlushSecsLeft : INT;    // countdown [s] before the SPX valve auto-opens

    tonFlush       : TON;    // delay before the flush (tFLUSH_DELAY)
    tonBlink       : TON;    // 0.5 s blink generator for the flashing buttons
    bBlinkPhase    : BOOL;
    bCleanPrev     : BOOL;   // clean-active on the previous scan (exit edge)

    i : INT;
	
	 // ---- water animation (spray strokes + clean flush) ----
    bWaterFlow : BOOL;                   // TRUE = stream visible
    abDrop     : ARRAY[0..3] OF BOOL;    // one flag per droplet, top -> bottom
    nDropIdx   : INT;                    // chaser position
    tonDrop    : TON;
    j          : INT;
END_VAR

VAR CONSTANT
    cGREEN  : DWORD := 16#FF46A758;   // open / auto / OK
    cGREY   : DWORD := 16#FF8A8F98;   // closed
    cRED    : DWORD := 16#FFE5484D;   // in transit / fault
    cYELLOW : DWORD := 16#FFF2C94C;   // manual
	cBLACK  : DWORD := 16#FF000000;

    // ---- clean-mode steps ----
    nCLEAN_OFF       : INT := 0;   // clean mode not active
    nCLEAN_READY     : INT := 1;   // entered clean; waiting for Start Clean
    nCLEAN_DRAIN     : INT := 2;   // pump runs until the tank reads ~0 %
    nCLEAN_ACK       : INT := 3;   // pump off; Close Drain + Add Water flash
    nCLEAN_REFILL    : INT := 4;   // acks done; wait level >= 20 % + Start Clean
    nCLEAN_FLUSHWAIT : INT := 5;   // 20 s countdown, then SPX auto-opens
    nCLEAN_FLUSH     : INT := 6;   // SPX open, pump flushes the pipes

    rCLEAN_EMPTY : REAL := 0.5;    // 'tank is 0' threshold [%]
    rCLEAN_FILL  : REAL := 20.0;   // refill minimum [%] - flush allowed at or above this
    tFLUSH_DELAY : TIME := T#20S;  // wait before the SPX valve auto-opens
	
	nDROP_COUNT : INT  := 6;         // droplets in the column (= abDrop size)
    nDROP_LIT   : INT  := 3;         // lit at once = visible stream length
    tDROP_STEP  : TIME := T#100MS;   // time per step -> fall speed
END_VAR

//==================================================================
// 1) NAV + STATE/ERROR TEXT
//==================================================================
FOR i := 0 TO 1 DO
    GVL_Nav.abNavActive[i] := (GVL_Nav.nPage = i);   // 0 = Spray, 1 = Machine Parameters
END_FOR

bFault := (MAIN.eState = E_SeqState.eFault) OR (MAIN.nErrorCode > 0);

CASE MAIN.eState OF
    E_SeqState.eIdle:         sStateText := 'Idle / circulation';
    E_SeqState.eDewater:      sStateText := 'T1 - dewater';
    E_SeqState.eSprayOpen:    sStateText := 'Spray - opening';
    E_SeqState.eSprayClose:   sStateText := 'Spray - closing';
    E_SeqState.eCloseDewater: sStateText := 'T5 - dewater / close';
ELSE
    sStateText := 'Fault';
END_CASE

CASE MAIN.nErrorCode OF
    0:  sErrorText := 'No fault';
    10: sErrorText := 'Piston not at P-close';
    20: sErrorText := 'SPX valve stuck (open)';
    21: sErrorText := 'SPX valve stuck (close)';
    30: sErrorText := 'Piston open timeout';
    40: sErrorText := 'Piston close timeout';
	50: sErrorText := 'SPX level high (>95%)';
	51: sErrorText := 'SPX level low (<5%)';
    99: sErrorText := 'Unknown state';
ELSE
    sErrorText := 'Fault';
END_CASE

// non-latching warnings (most relevant one)
IF GVL_Process.bLevelEmpty THEN
    sWarnText := 'SPX TANK EMPTY - pump off, mother held';
ELSIF GVL_Process.bWarnLevelLow THEN
    sWarnText := 'SPX level low (<20%)';
ELSIF GVL_Process.bWarnLevelHigh THEN
    sWarnText := 'SPX level high (>95%)';
ELSIF GVL_Process.bWarnBadSPX THEN
    sWarnText := 'Bad SPX pressure';
ELSIF GVL_Process.bWarnCircPress THEN
    sWarnText := 'Adjust circulation pressure';
ELSE
    sWarnText := '';
END_IF

//==================================================================
// 2) VALVE COLOURS   green = open, grey = closed, red = in transit
//==================================================================
// SPX valve - by the traffic-light feedback
IF GVL_IO.bSPXFullyOpen THEN
    cSPXValve := cGREEN;
ELSIF GVL_IO.bSPXFullyClose THEN
    cSPXValve := cGREY;
ELSE
    cSPXValve := cRED;                 // neither end -> moving
END_IF

// Circulation valve - the inverse of SPX
IF GVL_IO.bSPXFullyClose THEN
    cCircValve := cGREEN;              // SPX closed  -> circulation open
ELSIF GVL_IO.bSPXFullyOpen THEN
    cCircValve := cGREY;              // SPX open    -> circulation closed
ELSE
    cCircValve := cRED;
END_IF

// Air valve - by command (solenoid, no feedback)
IF GVL_IO.bAirValve THEN cAirValve := cGREEN; ELSE cAirValve := cGREY; END_IF

//==================================================================
// 3) PISTON LAMPS + MOLD LAMP + SPRAY MARKS
//==================================================================
IF GVL_IO.bPistonOpen  THEN cPistonOpen  := cGREEN; ELSE cPistonOpen  := cGREY; END_IF
IF GVL_IO.bPistonClosed THEN cPistonClose := cGREEN; ELSE cPistonClose := cGREY; END_IF

bMoldLamp := GVL_IO.bMoldAtSprayHigh;

// spray marks: piston off BOTH ends AND SPX + Air valves open
bSprayMarks := (NOT GVL_IO.bPistonOpen) AND (NOT GVL_IO.bPistonClosed)
            AND GVL_IO.bSPXValve AND GVL_IO.bAirValve;
			
//==================================================================
// 3b) WATER ANIMATION under the piston
//   Visible during the spray strokes (steps 20 / 30) and while the
//   clean sequence is flushing the pipes. nDropY repeats 0..spacing;
//   droplets placed one spacing apart read as a continuous stream.
//==================================================================
bWaterFlow := (MAIN.eState = E_SeqState.eSprayOpen)     // step 20
           OR (MAIN.eState = E_SeqState.eSprayClose)    // step 30
           OR (nCleanStep = nCLEAN_FLUSH);              // clean-mode flush

tonDrop(IN := bWaterFlow AND NOT tonDrop.Q, PT := tDROP_STEP);
IF NOT bWaterFlow THEN
    nDropIdx := 0;                       // always restart at the top
ELSIF tonDrop.Q THEN
    nDropIdx := (nDropIdx + 1) MOD nDROP_COUNT;
END_IF

FOR j := 0 TO nDROP_COUNT - 1 DO
    abDrop[j] := bWaterFlow
             AND (((j - nDropIdx + nDROP_COUNT) MOD nDROP_COUNT) < nDROP_LIT);
END_FOR

//==================================================================
// 4) MODE COLOUR / TEXT   manual = yellow, auto = green, fault = red
//==================================================================
IF bFault THEN
    cModeColor := cRED;    sModeText := 'FAULT';
ELSIF MAIN.bAutoMode THEN
    cModeColor := cGREEN;  sModeText := 'AUTO';
ELSE
    cModeColor := cYELLOW; sModeText := 'MANUAL';
END_IF

//------------------------------------------------------------------
// Readout colours - reuse the flags PRG_Process/MAIN already evaluate
//------------------------------------------------------------------
IF GVL_Process.bLevelEmpty THEN
    cLevel := cRED;                       // < rLevelEmpty -> pump stop / lockout
ELSIF GVL_Process.bWarnLevelLow OR GVL_Process.bWarnLevelHigh THEN
    cLevel := cYELLOW;
ELSE
    cLevel := cBLACK;
END_IF

IF GVL_Process.bWarnBadSPX THEN
    cSPXPress := cYELLOW;                 // last cycle's T3/T4 average off target
ELSE
    cSPXPress := cBLACK;
END_IF

//==================================================================
// 5) LIVE READOUTS
//==================================================================
rPumpHz      := GVL_IO.rPumpHz;
rSPXLevel    := GVL_IO.rSPXLevel;
rSPXPressure := GVL_IO.rSPXPressure;
rAirPressure := GVL_IO.rAirPressure;

//==================================================================
// 6) MANUAL MODE
//   Live only when AUTO is off and the sequence is idle. Buttons
//   toggle each actuator; MAIN applies bMan* while bManualActive.
//   While CLEAN MODE runs, the clean sequence (6b) owns the pump.
//   The pump follows the 'Pump speed' machine parameter
//   (GVL_Param.rPumpSpeedBase), so an Apply on the Params page takes
//   effect immediately here and in clean mode (6b).
//==================================================================
// mirror the machine parameter every scan - rManPumpHz has no HMI
// field of its own; the Params page is the single place to set it
rManPumpHz := GVL_Param.rPumpSpeedBase;

bManualActive := (NOT MAIN.bAutoMode) AND (MAIN.eState = E_SeqState.eIdle);

IF NOT bManualActive THEN
    bManAirValve    := FALSE;
    bManSPXValve    := FALSE;
    bManPistonOpen  := FALSE;
    bManPistonClose := FALSE;
ELSIF nCleanStep = nCLEAN_OFF THEN
    // manual pump setpoint drives the VFD directly (empty still wins)
    IF GVL_Process.bLevelEmpty THEN
        GVL_IO.rPumpHz := 0.0;
    ELSE
        GVL_IO.rPumpHz := rManPumpHz;
    END_IF
END_IF

//==================================================================
// 6b) CLEAN MODE   (manual only - button hidden otherwise)
//   READY:     operator opens the drain, presses Start Clean
//   DRAIN:     pump runs (empty lockout bypassed) until level ~0 %
//   ACK:       pump off; 'Close Drain' + 'Add Water' flash until
//              the operator presses each one
//   REFILL:    operator fills the tank to 20 % or more and closes
//              the fill valve; Start Clean accepted at level >= 20 %
//   FLUSHWAIT: 20 s countdown shown on the HMI...
//   FLUSH:     ...then the SPX valve is opened automatically (same
//              path as the manual SPX button) and the pump flushes
//              the spray pipes; when the tank runs dry the flush
//              stops and clean mode EXITS by itself
//   STOP CLEAN at any time stops everything and leaves clean mode.
//   NOTE: this runs AFTER PRG_Process in the task, so its rPumpHz
//   writes win the scan (same mechanism as the manual pump above).
//==================================================================
// ---- enter / stop ----
IF bBtnClean THEN
    IF nCleanStep = nCLEAN_OFF THEN
        IF bManualActive THEN
            nCleanStep := nCLEAN_READY;
            bDrainAck  := FALSE;
            bWaterAck  := FALSE;
        END_IF
    ELSE
        // STOP CLEAN - stop whatever the sequence is doing
        nCleanStep     := nCLEAN_OFF;
        bManSPXValve   := FALSE;     // close the SPX valve if flushing
        GVL_IO.rPumpHz := 0.0;       // normal manual logic resumes next scan
    END_IF
END_IF

// leaving manual (fault / sequence running) aborts clean mode
IF (nCleanStep <> nCLEAN_OFF) AND NOT bManualActive THEN
    nCleanStep     := nCLEAN_OFF;
    GVL_IO.rPumpHz := 0.0;
END_IF

bCleanActive := (nCleanStep <> nCLEAN_OFF);

// 0.5 s blink generator for the flashing prompt buttons
tonBlink(IN := NOT tonBlink.Q, PT := T#500MS);
IF tonBlink.Q THEN
    bBlinkPhase := NOT bBlinkPhase;
END_IF

CASE nCleanStep OF

    nCLEAN_OFF:
        tonFlush(IN := FALSE);
        bDrainFlash  := FALSE;
        bWaterFlash  := FALSE;
        sCleanStatus := '';

    nCLEAN_READY:
        // circulation keeps running at the manual setpoint until drain starts
        IF GVL_Process.bLevelEmpty THEN
            GVL_IO.rPumpHz := 0.0;
        ELSE
            GVL_IO.rPumpHz := rManPumpHz;
        END_IF
        sCleanStatus := 'Open the drain, then press Start Clean';
        IF bBtnStartClean THEN
            nCleanStep := nCLEAN_DRAIN;
        END_IF

    nCLEAN_DRAIN:
        // pump keeps running below the normal empty lockout - the goal IS 0 %
        GVL_IO.rPumpHz := rManPumpHz;
        sCleanStatus   := 'Draining tank...';
        IF GVL_IO.rSPXLevel <= rCLEAN_EMPTY THEN
            GVL_IO.rPumpHz := 0.0;
            bDrainAck  := FALSE;
            bWaterAck  := FALSE;
            nCleanStep := nCLEAN_ACK;
        END_IF

    nCLEAN_ACK:
        GVL_IO.rPumpHz := 0.0;
        sCleanStatus   := 'Tank empty - close the drain and add water';
        IF bBtnCloseDrain THEN bDrainAck := TRUE; END_IF
        IF bBtnAddWater  THEN bWaterAck := TRUE; END_IF
        bDrainFlash := (NOT bDrainAck) AND bBlinkPhase;
        bWaterFlash := (NOT bWaterAck) AND bBlinkPhase;
        IF bDrainAck AND bWaterAck THEN
            bDrainFlash := FALSE;
            bWaterFlash := FALSE;
            nCleanStep  := nCLEAN_REFILL;
        END_IF

    nCLEAN_REFILL:
        GVL_IO.rPumpHz := 0.0;
        IF GVL_IO.rSPXLevel >= rCLEAN_FILL THEN
            sCleanStatus := 'Ready - press Start Clean to flush the pipes';
            IF bBtnStartClean THEN
                tonFlush(IN := FALSE);           // make sure the timer restarts
                nCleanStep := nCLEAN_FLUSHWAIT;
            END_IF
        ELSE
            sCleanStatus := 'Fill the tank to 20% or more, then close the fill valve';
            // Start Clean is ignored until the tank holds at least 20 %
        END_IF

    nCLEAN_FLUSHWAIT:
        // circulate the fresh water while the countdown runs
        GVL_IO.rPumpHz := rManPumpHz;
        tonFlush(IN := TRUE, PT := tFLUSH_DELAY);
        nFlushSecsLeft := DINT_TO_INT(
            (TIME_TO_DINT(tFLUSH_DELAY) - TIME_TO_DINT(tonFlush.ET)) / 1000);
        IF nFlushSecsLeft < 0 THEN nFlushSecsLeft := 0; END_IF
        sCleanStatus := CONCAT(CONCAT('Opening SPX valve in ',
                        INT_TO_STRING(nFlushSecsLeft)), ' s');
        IF tonFlush.Q THEN
            tonFlush(IN := FALSE);
            bManSPXValve := TRUE;    // auto-'press' the manual SPX-valve button
            nCleanStep   := nCLEAN_FLUSH;
        END_IF

    nCLEAN_FLUSH:
        // pump pushes water through the open SPX line
        IF GVL_IO.rSPXLevel <= rCLEAN_EMPTY THEN
            // tank dry -> flush finished: stop and leave clean mode by itself
            GVL_IO.rPumpHz := 0.0;
            bManSPXValve   := FALSE;         // close the SPX valve
            nCleanStep     := nCLEAN_OFF;
        ELSE
            GVL_IO.rPumpHz := rManPumpHz;
            sCleanStatus   := 'Flushing pipes - press Stop Clean to finish';
        END_IF

END_CASE

//------------------------------------------------------------------
// post-clean empty latch: leaving clean mode with a dry tank (auto
// flush-complete OR Stop Clean mid-way) must not latch the level-LOW
// fault in MAIN. Suppressed until the tank is refilled above 5 %.
//------------------------------------------------------------------
IF bCleanPrev AND (nCleanStep = nCLEAN_OFF)
   AND (GVL_IO.rSPXLevel < GVL_Param.rLevelEmpty) THEN
    bPostCleanEmpty := TRUE;
END_IF
IF GVL_IO.rSPXLevel >= GVL_Param.rLevelEmpty THEN
    bPostCleanEmpty := FALSE;    // refilled -> normal protection resumes
END_IF
bCleanPrev := (nCleanStep <> nCLEAN_OFF);

// clean-button label follows the mode
IF bCleanActive THEN
    sCleanBtnText := 'STOP CLEAN';
ELSE
    sCleanBtnText := 'CLEAN MODE';
END_IF

//==================================================================
// 7) CONSUME COMMAND BITS
//   MAIN read them at the top of this scan; clearing here means the
//   HMI button only has to write TRUE once per press. The clean
//   buttons were consumed by section 6b just above.
//==================================================================
bCmdAuto  := FALSE;
bCmdReset := FALSE;
bBtnClean      := FALSE;
bBtnStartClean := FALSE;
bBtnCloseDrain := FALSE;
bBtnAddWater   := FALSE;

END_PROGRAM

// ---- POUs/PRG_Process.TcPOU
PROGRAM PRG_Process
//==================================================================
// PROCESS SUPERVISION  (spec slide 10 - "general")
//   1) SPX tank level monitoring (warnings + empty lockout)
//   2) gear-pump speed: P-only control, updated once per cycle
//   3) circulation-pressure sanity check
//
//   *** The pump gain/limits are the values the spec left open
//       ("?? find the Hz amount"). They live in GVL_Param and must be
//       tuned on the machine - the STRUCTURE here is complete. ***
//==================================================================
VAR
    rtCycleEnd : R_TRIG;   // fires when a spray cycle finishes (busy 1 -> 0)
    bWasBusy   : BOOL;     // previous-scan bSprayBusy
END_VAR

//------------------------------------------------------------------
// 1) SPX TANK LEVEL MONITORING
//------------------------------------------------------------------
GVL_Process.bWarnLevelHigh := GVL_IO.rSPXLevel > GVL_Param.rLevelHigh;   // > 95%
GVL_Process.bWarnLevelLow  := GVL_IO.rSPXLevel < GVL_Param.rLevelLow;    // < 20%
GVL_Process.bLevelEmpty    := GVL_IO.rSPXLevel < GVL_Param.rLevelEmpty;  // < 5%  -> halt

//------------------------------------------------------------------
// 2) GEAR-PUMP SPEED  -  P-only, updated at the END of each cycle
//   End of cycle = bSprayBusy falls 1 -> 0 after a normal release.
//   On a fault MAIN drops bSprayBusy too, so gate on NOT bError.
//------------------------------------------------------------------
rtCycleEnd(CLK := bWasBusy AND NOT GVL_IO.bSprayBusy);
bWasBusy := GVL_IO.bSprayBusy;

IF rtCycleEnd.Q AND NOT MAIN.bError THEN
    // combined spray-pressure average for the cycle
    GVL_Process.rSPXAvg := (GVL_Process.rSPXAvgT3 + GVL_Process.rSPXAvgT4) * 0.5;

    // P correction with deadband:
    //   measured too HIGH -> slow the pump down
    //   measured too LOW  -> speed the pump up
    // "double the difference" from the spec is captured by rPumpKp (TBD).
    IF (GVL_Process.rSPXAvg - GVL_Param.rSPXPressureTarget) > GVL_Param.rPumpDeadband THEN
        GVL_IO.rPumpHz := GVL_IO.rPumpHz
                        - GVL_Param.rPumpKp * (GVL_Process.rSPXAvg - GVL_Param.rSPXPressureTarget);
    ELSIF (GVL_Param.rSPXPressureTarget - GVL_Process.rSPXAvg) > GVL_Param.rPumpDeadband THEN
        GVL_IO.rPumpHz := GVL_IO.rPumpHz
                        + GVL_Param.rPumpKp * (GVL_Param.rSPXPressureTarget - GVL_Process.rSPXAvg);
    END_IF

    // clamp to the configured pump window
    GVL_IO.rPumpHz := LIMIT(GVL_Param.rPumpHzMin, GVL_IO.rPumpHz, GVL_Param.rPumpHzMax);

    // circulation-pressure sanity: spray avg vs circulation avg
    GVL_Process.bWarnCircPress :=
        ABS(GVL_Process.rSPXAvg - GVL_Process.rSPXAvgCirc) > GVL_Param.rCircPressTol;
END_IF

// initialise the pump to the base setpoint on the first scan (or after a refill)
IF GVL_IO.rPumpHz <= 0.0 AND NOT GVL_Process.bLevelEmpty THEN
    GVL_IO.rPumpHz := GVL_Param.rPumpSpeedBase;
END_IF

//------------------------------------------------------------------
// 3) TANK-EMPTY LOCKOUT  -  stop the pump (release is blocked in MAIN)
//------------------------------------------------------------------
IF GVL_Process.bLevelEmpty THEN
    GVL_IO.rPumpHz := 0.0;
END_IF

END_PROGRAM

// ---- POUs/PRG_Params.TcPOU
PROGRAM PRG_Params
//==================================================================
// MACHINE PARAMETERS SCREEN  (page 1)
//   The operator edits the *Edit* copies (tap a value -> numeric keypad);
//   LOAD pulls the live values in, APPLY writes them to GVL_Param.
//   RESET loads the factory defaults (GVL_Param.cDef*) into the edit
//   copies and then runs the EXACT same gate as APPLY (idle + sanity).
//   The RESET button is only visible in manual mode on the HMI.
//
//   The time fields are edited as REAL SECONDS (so the HMI keypad shows
//   plain decimals: 4, 0.5, 3.0, 10) and converted to TIME on apply.
//   The HMI groups two pairs into one value each:
//     "T2 & T6" -> rEditValveMax_s   (writes both watchdogs)
//     "T3 & T4" -> rEditSprayTime_s   (writes both watchdogs)
//   APPLY is only accepted while the sequence is idle.
//
//   For the event logger (PRG_FileLogger reads these on bMsgTrig):
//     bLastApplyOk  - result of the last Apply/Reset press
//     bLastWasReset - that press came from the RESET button
//     sChangeList   - ONLY the params that changed, 'old->new' each;
//                     EMPTY if identical values were applied (not logged)
//==================================================================
VAR
    // ---- editable copies in SECONDS (bound to the HMI keypad fields) ----
    rEditDewater_s    : REAL;   // T1 : Dewater time            [s]
    rEditValveMax_s   : REAL;   // T2 & T6 : valve max open/close[s]
    rEditSprayTime_s  : REAL;   // T3 & T4 : max spraying time   [s]
    rEditSPXDewater_s : REAL;   // T5 : SPX Dewater time         [s]
    rEditPressTarget  : REAL;   // SPX Pressure target           [bar]
    rEditPumpSpeed    : REAL;   // Pump speed                    [Hz]

    // ---- buttons ----
    bBtnApply : BOOL;          // "Apply" (write edits to GVL_Param)
    bBtnLoad  : BOOL;          // "Reload" (discard edits, pull live values)
    bBtnReset : BOOL;          // "Reset defaults" (manual mode only on the HMI)

    // ---- status ----
    bApplyAllowed : BOOL;      // TRUE while edits may be applied (idle)
    sParamStatus  : STRING := 'Ready';
    bInit         : BOOL;      // first-scan load

    // ---- info for the event logger (PRG_FileLogger) ----
    bLastApplyOk  : BOOL;          // result of the last Apply/Reset press
    bLastWasReset : BOOL;          // TRUE if that press was the RESET button
    sChangeList   : STRING(255);   // changed params only, old->new

    // ---- 5 s message window (drives HMI message visibility) ----
    bMsgVisible : BOOL;        // TRUE for 5 s after Apply, then FALSE
    bMsgTrig    : BOOL;        // one-scan trigger (Apply/Reset pressed)
    tonMsg      : TON;         // 5 s display timer

    // ---- internal ----
    bResetActive : BOOL;       // current press came from RESET
    tNewT1  : TIME;            // converted-once new values (also used
    tNewT26 : TIME;            //  for the changed/unchanged comparison)
    tNewT34 : TIME;
    tNewT5  : TIME;
    rOldVal : REAL;            // scratch: old value in display units
END_VAR

VAR CONSTANT
    rMS_PER_S  : REAL := 1000.0;
    tMSG_SHOW  : TIME := T#3S;   // how long the status / banner stays visible
END_VAR

// On the first scan, pull the live parameters into the edit copies.
bMsgTrig := FALSE;   // reset the one-scan message trigger

IF NOT bInit THEN
    bInit    := TRUE;
    bBtnLoad := TRUE;
END_IF

// Parameters may only be applied while the sequence is idle.
bApplyAllowed := (MAIN.eState = E_SeqState.eIdle);

// ---- LOAD: live (TIME) -> edit copies (REAL seconds) ----
IF bBtnLoad THEN
    bBtnLoad := FALSE;
    rEditDewater_s    := DINT_TO_REAL(TIME_TO_DINT(GVL_Param.tDewaterTime))     / rMS_PER_S;
    rEditValveMax_s   := DINT_TO_REAL(TIME_TO_DINT(GVL_Param.tSPXMaxOpenTime))  / rMS_PER_S;
    rEditSprayTime_s  := DINT_TO_REAL(TIME_TO_DINT(GVL_Param.tSprayOpenTime))   / rMS_PER_S;
    rEditSPXDewater_s := DINT_TO_REAL(TIME_TO_DINT(GVL_Param.tSPXDewaterTime))  / rMS_PER_S;
    rEditPressTarget  := GVL_Param.rSPXPressureTarget;
    rEditPumpSpeed    := GVL_Param.rPumpSpeedBase;
    sParamStatus      := 'Loaded';
END_IF

// ---- RESET: factory defaults -> edit copies, then the SAME path as APPLY ----
//   (the HMI shows this button only in manual mode; the idle gate and the
//    sanity checks below still run exactly as for a normal Apply)
IF bBtnReset THEN
    bBtnReset := FALSE;
    rEditDewater_s    := DINT_TO_REAL(TIME_TO_DINT(GVL_Param.cDefDewaterTime))    / rMS_PER_S;
    rEditValveMax_s   := DINT_TO_REAL(TIME_TO_DINT(GVL_Param.cDefValveMaxTime))   / rMS_PER_S;
    rEditSprayTime_s  := DINT_TO_REAL(TIME_TO_DINT(GVL_Param.cDefSprayTime))      / rMS_PER_S;
    rEditSPXDewater_s := DINT_TO_REAL(TIME_TO_DINT(GVL_Param.cDefSPXDewaterTime)) / rMS_PER_S;
    rEditPressTarget  := GVL_Param.cDefPressTarget;
    rEditPumpSpeed    := GVL_Param.cDefPumpSpeed;
    bResetActive := TRUE;
    bBtnApply    := TRUE;    // fall through into the apply gate below
END_IF

// ---- APPLY: edit copies (REAL seconds) -> live (TIME), idle + sanity ----
IF bBtnApply THEN
    bBtnApply := FALSE;
    bMsgTrig  := TRUE;     // show the status (and the manual banner) for 3 s
    IF NOT bApplyAllowed THEN
        sParamStatus := 'Rejected: sequence not idle';
        bLastApplyOk := FALSE;
    ELSIF (rEditDewater_s <= 0.0) OR (rEditValveMax_s <= 0.0) OR (rEditSprayTime_s <= 0.0)
       OR (rEditSPXDewater_s <= 0.0) OR (rEditPumpSpeed <= 0.0) THEN
        sParamStatus := 'Rejected: values must be > 0';
        bLastApplyOk := FALSE;
    ELSE
        // seconds -> milliseconds -> TIME (converted once, reused below)
        tNewT1  := DINT_TO_TIME(REAL_TO_DINT(rEditDewater_s    * rMS_PER_S));
        tNewT26 := DINT_TO_TIME(REAL_TO_DINT(rEditValveMax_s   * rMS_PER_S));
        tNewT34 := DINT_TO_TIME(REAL_TO_DINT(rEditSprayTime_s  * rMS_PER_S));
        tNewT5  := DINT_TO_TIME(REAL_TO_DINT(rEditSPXDewater_s * rMS_PER_S));

        // ---- change list: ONLY the params that actually change (old->new) ----
        sChangeList := '';
        IF tNewT1 <> GVL_Param.tDewaterTime THEN
            rOldVal := DINT_TO_REAL(TIME_TO_DINT(GVL_Param.tDewaterTime)) / rMS_PER_S;
            sChangeList := CONCAT(sChangeList, 'T1 ');
            sChangeList := CONCAT(sChangeList, LREAL_TO_FMTSTR(REAL_TO_LREAL(rOldVal), 1, TRUE));
            sChangeList := CONCAT(sChangeList, '->');
            sChangeList := CONCAT(sChangeList, LREAL_TO_FMTSTR(REAL_TO_LREAL(rEditDewater_s), 1, TRUE));
            sChangeList := CONCAT(sChangeList, 's, ');
        END_IF
        IF tNewT26 <> GVL_Param.tSPXMaxOpenTime THEN     // T2 & T6 always written as a pair
            rOldVal := DINT_TO_REAL(TIME_TO_DINT(GVL_Param.tSPXMaxOpenTime)) / rMS_PER_S;
            sChangeList := CONCAT(sChangeList, 'T2/T6 ');
            sChangeList := CONCAT(sChangeList, LREAL_TO_FMTSTR(REAL_TO_LREAL(rOldVal), 1, TRUE));
            sChangeList := CONCAT(sChangeList, '->');
            sChangeList := CONCAT(sChangeList, LREAL_TO_FMTSTR(REAL_TO_LREAL(rEditValveMax_s), 1, TRUE));
            sChangeList := CONCAT(sChangeList, 's, ');
        END_IF
        IF tNewT34 <> GVL_Param.tSprayOpenTime THEN      // T3 & T4 always written as a pair
            rOldVal := DINT_TO_REAL(TIME_TO_DINT(GVL_Param.tSprayOpenTime)) / rMS_PER_S;
            sChangeList := CONCAT(sChangeList, 'T3/T4 ');
            sChangeList := CONCAT(sChangeList, LREAL_TO_FMTSTR(REAL_TO_LREAL(rOldVal), 1, TRUE));
            sChangeList := CONCAT(sChangeList, '->');
            sChangeList := CONCAT(sChangeList, LREAL_TO_FMTSTR(REAL_TO_LREAL(rEditSprayTime_s), 1, TRUE));
            sChangeList := CONCAT(sChangeList, 's, ');
        END_IF
        IF tNewT5 <> GVL_Param.tSPXDewaterTime THEN
            rOldVal := DINT_TO_REAL(TIME_TO_DINT(GVL_Param.tSPXDewaterTime)) / rMS_PER_S;
            sChangeList := CONCAT(sChangeList, 'T5 ');
            sChangeList := CONCAT(sChangeList, LREAL_TO_FMTSTR(REAL_TO_LREAL(rOldVal), 1, TRUE));
            sChangeList := CONCAT(sChangeList, '->');
            sChangeList := CONCAT(sChangeList, LREAL_TO_FMTSTR(REAL_TO_LREAL(rEditSPXDewater_s), 1, TRUE));
            sChangeList := CONCAT(sChangeList, 's, ');
        END_IF
        IF rEditPressTarget <> GVL_Param.rSPXPressureTarget THEN
            sChangeList := CONCAT(sChangeList, 'Ptgt ');
            sChangeList := CONCAT(sChangeList, LREAL_TO_FMTSTR(REAL_TO_LREAL(GVL_Param.rSPXPressureTarget), 2, TRUE));
            sChangeList := CONCAT(sChangeList, '->');
            sChangeList := CONCAT(sChangeList, LREAL_TO_FMTSTR(REAL_TO_LREAL(rEditPressTarget), 2, TRUE));
            sChangeList := CONCAT(sChangeList, 'bar, ');
        END_IF
        IF rEditPumpSpeed <> GVL_Param.rPumpSpeedBase THEN
            sChangeList := CONCAT(sChangeList, 'Pump ');
            sChangeList := CONCAT(sChangeList, LREAL_TO_FMTSTR(REAL_TO_LREAL(GVL_Param.rPumpSpeedBase), 1, TRUE));
            sChangeList := CONCAT(sChangeList, '->');
            sChangeList := CONCAT(sChangeList, LREAL_TO_FMTSTR(REAL_TO_LREAL(rEditPumpSpeed), 1, TRUE));
            sChangeList := CONCAT(sChangeList, 'Hz, ');
        END_IF
        IF sChangeList <> '' THEN
            sChangeList := LEFT(sChangeList, LEN(sChangeList) - 2);   // drop trailing ', '
        END_IF

        // ---- write ----
        GVL_Param.tDewaterTime       := tNewT1;
        GVL_Param.tSPXMaxOpenTime    := tNewT26;   // T2
        GVL_Param.tSPXMaxCloseTime   := tNewT26;   // T6 (shares value)
        GVL_Param.tSprayOpenTime     := tNewT34;   // T3
        GVL_Param.tSprayCloseTime    := tNewT34;   // T4 (shares value)
        GVL_Param.tSPXDewaterTime    := tNewT5;
        GVL_Param.rSPXPressureTarget := rEditPressTarget;
        GVL_Param.rPumpSpeedBase     := rEditPumpSpeed;

        bLastApplyOk := TRUE;
        IF sChangeList = '' THEN
            sParamStatus := 'No changes';        // accepted, nothing to do -> NOT logged
        ELSIF bResetActive THEN
            sParamStatus := 'Reset to defaults';
        ELSE
            sParamStatus := 'Applied';
        END_IF
    END_IF
    bLastWasReset := bResetActive;   // tell the logger where this press came from
    bResetActive  := FALSE;
END_IF

// ---- 5 s message window ----
//   bMsgVisible goes TRUE on Apply and stays TRUE for tMSG_SHOW, then drops.
//   The HMI binds the status text / manual banner "Invisible" to NOT this flag.
IF bMsgTrig THEN
    bMsgVisible := TRUE;
    tonMsg(IN := FALSE);              // restart the window on each press
END_IF
tonMsg(IN := bMsgVisible, PT := tMSG_SHOW);
IF tonMsg.Q THEN
    bMsgVisible := FALSE;
END_IF

END_PROGRAM

// ---- POUs/PRG_FileLogger.TcPOU
PROGRAM PRG_FileLogger
//==================================================================
// MACHINE EVENT LOGGER (observer)
//   Watches MAIN / GVL_Process / PRG_Spray / PRG_Params and logs one
//   line per EVENT. By design there are NO duration measurements
//   (no "step X took Y s") - only what happened and when.
//
//   File: <GVL_Param.sLogDir>/machine_events_YYYY-MM.log
//         (one file per month; legend header on boot/rollover)
//   Tags: [.] INFO   [!] WARN   [X] ERROR
//
//   Severity map:
//     [X] ERROR - latched sequence faults          (MAIN.nErrorCode)
//     [!] WARN  - process warnings, cycle aborts,  (GVL_Process.bWarn*,
//                 parameter changes (applied/reset)  AUTO abort, PRG_Params)
//                 and rejected parameter writes
//     [.] INFO  - boot, AUTO/MANUAL, manual presses, cycle start/
//                 complete, fault reset, state changes, param snapshots
//
//   PARAM SNAPSHOT (for the Grafana dashboard): one INFO line with ALL
//   current machine parameters ('Params snapshot: T1=... Pump=...Hz')
//   is written at boot, after every accepted Apply/Reset, and every
//   tSnapBeat (heartbeat) so the dashboard's lookback window always
//   finds a fresh one. Grafana extracts the numbers with regexp+unwrap.
//
//   All detection lives HERE - no other POU was touched. If you ever
//   want to log directly from another POU (same task!), you can:
//       PRG_FileLogger.fbLog.Info('my message');
//
//   Log file health: watch fbLog.nFailCount / nDropped / nLastErrId /
//   sLastPath online if the file stays empty (Linux: permissions!).
//==================================================================
VAR
    fbLog : FB_EventLog := (sBaseName := 'machine_events');

    // ---- one-shot startup ----
    bStartupLogged : BOOL;

    // ---- previous-scan copies for change detection ----
    ePrevState : E_SeqState := E_SeqState.eIdle;
    bPrevAuto  : BOOL;
    bPrevSim   : BOOL := TRUE;     // matches SIM_Plant.bSimEnable init -> no ghost line at boot
    nLastFault : INT;              // captured on fault entry (MAIN clears nErrorCode on reset)

    // ---- manual-mode presses ----
    bPrevManAir    : BOOL;
    bPrevManSPX    : BOOL;
    bPrevManPOpen  : BOOL;
    bPrevManPClose : BOOL;
    bPrevManPump   : BOOL;
    rPrevManHz     : REAL := 15.0; // matches PRG_Spray init -> no ghost line at boot

    // ---- process-warning edges + chatter cooldowns ----
    // (cooldown only for the analog level thresholds, where the value
    //  can hover at the limit; the per-cycle warnings are edge-only)
    rtLevelLow   : R_TRIG;   tonCoolLow   : TON;   bCoolLow   : BOOL;
    rtLevelHigh  : R_TRIG;   tonCoolHigh  : TON;   bCoolHigh  : BOOL;
    rtLevelEmpty : R_TRIG;   tonCoolEmpty : TON;   bCoolEmpty : BOOL;
    rtBadSPX     : R_TRIG;
    rtCircPress  : R_TRIG;
    tCooldown    : TIME := T#60S;  // min spacing per level warning

    // ---- HMI / parameter events ----
    rtParamMsg : R_TRIG;

    // ---- parameter snapshot (full current values, for the dashboard) ----
    bSnapReq    : BOOL;            // one-shot: write a snapshot this scan
    tonSnapBeat : TON;             // heartbeat -> Grafana lookback always hits
    tSnapBeat   : TIME := T#6H;    // snapshot spacing (4 lines/day)

    // ---- scratch line builder ----
    sTxt : STRING(255);
END_VAR

//------------------------------------------------------------------
// 0) STARTUP  (once, as soon as the local clock is valid)
//------------------------------------------------------------------
IF NOT bStartupLogged AND fbLog.bTimeValid THEN
    bStartupLogged := TRUE;
    fbLog.Info('=== PLC application started ===');
    IF SIM_Plant.bSimEnable THEN
        fbLog.Warn('SIMULATION mode active - I/O is simulated, not real hardware');
    END_IF
    bSnapReq := TRUE;              // boot -> log the full parameter set
END_IF

//------------------------------------------------------------------
// 1) SEQUENCE STATE CHANGES  (faults, resets, cycle start/complete)
//------------------------------------------------------------------
IF MAIN.eState <> ePrevState THEN

    IF MAIN.eState = E_SeqState.eFault THEN
        // ---------- [X] fault raised ----------
        nLastFault := MAIN.nErrorCode;
        sTxt := 'FAULT ';
        sTxt := CONCAT(sTxt, INT_TO_STRING(MAIN.nErrorCode));
        sTxt := CONCAT(sTxt, ': ');
        CASE MAIN.nErrorCode OF
            10: sTxt := CONCAT(sTxt, 'piston not at P-close');
            20: sTxt := CONCAT(sTxt, 'SPX valve stuck - never Fully Open (T2)');
            21: sTxt := CONCAT(sTxt, 'SPX valve stuck - never Fully Close (T6)');
            30: sTxt := CONCAT(sTxt, 'piston opening stroke timeout (T3)');
            40: sTxt := CONCAT(sTxt, 'piston closing stroke timeout (T4)');
            50: sTxt := CONCAT(sTxt, 'SPX level HIGH');
            51: sTxt := CONCAT(sTxt, 'SPX level EMPTY');
        ELSE
            sTxt := CONCAT(sTxt, 'unknown state');
        END_CASE
        sTxt := CONCAT(sTxt, ' (in ');
        sTxt := CONCAT(sTxt, TO_STRING(ePrevState));
        sTxt := CONCAT(sTxt, ', level ');
        sTxt := CONCAT(sTxt, LREAL_TO_FMTSTR(REAL_TO_LREAL(GVL_IO.rSPXLevel), 1, TRUE));
        sTxt := CONCAT(sTxt, ' %) - outputs safe, AUTO dropped');
        fbLog.Error(sTxt);

    ELSIF ePrevState = E_SeqState.eFault AND MAIN.eState = E_SeqState.eIdle THEN
        // ---------- [.] fault reset by operator ----------
        sTxt := 'Fault reset by operator (was FAULT ';
        sTxt := CONCAT(sTxt, INT_TO_STRING(nLastFault));
        sTxt := CONCAT(sTxt, ')');
        fbLog.Info(sTxt);

    ELSIF ePrevState = E_SeqState.eIdle AND MAIN.eState = E_SeqState.eDewater THEN
        // ---------- [.] spray cycle started (mother handshake accepted) ----------
        sTxt := 'Spray cycle started (SPX level ';
        sTxt := CONCAT(sTxt, LREAL_TO_FMTSTR(REAL_TO_LREAL(GVL_IO.rSPXLevel), 1, TRUE));
        sTxt := CONCAT(sTxt, ' %, pump ');
        sTxt := CONCAT(sTxt, LREAL_TO_FMTSTR(REAL_TO_LREAL(GVL_IO.rPumpHz), 1, TRUE));
        sTxt := CONCAT(sTxt, ' Hz)');
        fbLog.Info(sTxt);

    ELSIF ePrevState = E_SeqState.eCloseDewater AND MAIN.eState = E_SeqState.eIdle THEN
        // ---------- [.] spray cycle completed ----------
        // (PRG_Process already updated the averages + pump correction this
        //  same scan - it runs before this program in MAIN's call list)
        sTxt := 'Spray cycle completed (SPX avg T3 ';
        sTxt := CONCAT(sTxt, LREAL_TO_FMTSTR(REAL_TO_LREAL(GVL_Process.rSPXAvgT3), 2, TRUE));
        sTxt := CONCAT(sTxt, ' / T4 ');
        sTxt := CONCAT(sTxt, LREAL_TO_FMTSTR(REAL_TO_LREAL(GVL_Process.rSPXAvgT4), 2, TRUE));
        sTxt := CONCAT(sTxt, ' bar, pump -> ');
        sTxt := CONCAT(sTxt, LREAL_TO_FMTSTR(REAL_TO_LREAL(GVL_IO.rPumpHz), 1, TRUE));
        sTxt := CONCAT(sTxt, ' Hz)');
        fbLog.Info(sTxt);

    ELSIF GVL_Param.bLogStateChanges THEN
        // ---------- [.] any other transition (verbose, switchable) ----------
        sTxt := 'State: ';
        sTxt := CONCAT(sTxt, TO_STRING(ePrevState));
        sTxt := CONCAT(sTxt, ' -> ');
        sTxt := CONCAT(sTxt, TO_STRING(MAIN.eState));
        fbLog.Info(sTxt);
    END_IF
END_IF

//------------------------------------------------------------------
// 2) AUTO / MANUAL  (before updating ePrevState - the abort message
//    uses it to know whether a cycle was running)
//------------------------------------------------------------------
IF MAIN.bAutoMode AND NOT bPrevAuto THEN
    fbLog.Info('AUTO armed by operator');
ELSIF NOT MAIN.bAutoMode AND bPrevAuto AND NOT MAIN.bError THEN
    // (a fault also drops AUTO, but that's already in the [X] line)
    IF ePrevState <> E_SeqState.eIdle AND ePrevState <> E_SeqState.eFault THEN
        sTxt := 'AUTO stopped by operator - running cycle ABORTED to idle (was in ';
        sTxt := CONCAT(sTxt, TO_STRING(ePrevState));
        sTxt := CONCAT(sTxt, ')');
        fbLog.Warn(sTxt);
    ELSE
        fbLog.Info('AUTO stopped by operator -> MANUAL');
    END_IF
END_IF
bPrevAuto  := MAIN.bAutoMode;
ePrevState := MAIN.eState;

//------------------------------------------------------------------
// 2b) MANUAL PRESSES  (brief one-liners; only while manual is live.
//     PRG_Spray force-clears the flags on manual exit - not logged.)
//------------------------------------------------------------------
IF PRG_Spray.bManualActive THEN
    IF PRG_Spray.bManAirValve <> bPrevManAir THEN
        IF PRG_Spray.bManAirValve THEN fbLog.Info('MAN: Air ON');
        ELSE fbLog.Info('MAN: Air OFF'); END_IF
    END_IF
    IF PRG_Spray.bManSPXValve <> bPrevManSPX THEN
        IF PRG_Spray.bManSPXValve THEN fbLog.Info('MAN: SPX ON');
        ELSE fbLog.Info('MAN: SPX OFF'); END_IF
    END_IF
    IF PRG_Spray.bManPistonOpen <> bPrevManPOpen THEN
        IF PRG_Spray.bManPistonOpen THEN fbLog.Info('MAN: Piston-open sol ON');
        ELSE fbLog.Info('MAN: Piston-open sol OFF'); END_IF
    END_IF
    IF PRG_Spray.bManPistonClose <> bPrevManPClose THEN
        IF PRG_Spray.bManPistonClose THEN fbLog.Info('MAN: Piston-close sol ON');
        ELSE fbLog.Info('MAN: Piston-close sol OFF'); END_IF
    END_IF
    IF PRG_Spray.bManPump <> bPrevManPump THEN
        IF PRG_Spray.bManPump THEN fbLog.Info('MAN: Pump RUN');
        ELSE fbLog.Info('MAN: Pump STOP'); END_IF
    END_IF
    IF ABS(PRG_Spray.rManPumpHz - rPrevManHz) > 0.05 THEN
        sTxt := 'MAN: Pump ';
        sTxt := CONCAT(sTxt, LREAL_TO_FMTSTR(REAL_TO_LREAL(PRG_Spray.rManPumpHz), 1, TRUE));
        sTxt := CONCAT(sTxt, ' Hz');
        fbLog.Info(sTxt);
    END_IF
END_IF
// sync prev copies every scan -> no ghost edges when re-entering manual
bPrevManAir    := PRG_Spray.bManAirValve;
bPrevManSPX    := PRG_Spray.bManSPXValve;
bPrevManPOpen  := PRG_Spray.bManPistonOpen;
bPrevManPClose := PRG_Spray.bManPistonClose;
bPrevManPump   := PRG_Spray.bManPump;
rPrevManHz     := PRG_Spray.rManPumpHz;

//------------------------------------------------------------------
// 2c) SIM / REAL SOURCE SWITCH  (SIM_Plant.bSimEnable - HMI button)
//     Deserves its own line: every figure in the messages around it -
//     level, SPX/air pressure, pump Hz - changes meaning with this
//     flag, so a log read after the fact must say which source was
//     live. Gated on bStartupLogged: the boot state is reported by
//     section 0, and this must not repeat it as a "switch".
//------------------------------------------------------------------
IF bStartupLogged AND (SIM_Plant.bSimEnable <> bPrevSim) THEN
    IF SIM_Plant.bSimEnable THEN
        fbLog.Warn('Source -> SIMULATION: readouts are simulated, not measured');
    ELSE
        fbLog.Info('Source -> REAL I/O: simulated inputs released');
    END_IF
END_IF
bPrevSim := SIM_Plant.bSimEnable;

//------------------------------------------------------------------
// 3) PROCESS WARNINGS  (non-latching flags from GVL_Process)
//------------------------------------------------------------------
// -- SPX level low (< rLevelLow) --
tonCoolLow(IN := bCoolLow, PT := tCooldown);
IF tonCoolLow.Q THEN bCoolLow := FALSE; END_IF
rtLevelLow(CLK := GVL_Process.bWarnLevelLow);
IF rtLevelLow.Q AND NOT bCoolLow THEN
    bCoolLow := TRUE;
    sTxt := 'SPX level low: ';
    sTxt := CONCAT(sTxt, LREAL_TO_FMTSTR(REAL_TO_LREAL(GVL_IO.rSPXLevel), 1, TRUE));
    sTxt := CONCAT(sTxt, ' % (limit ');
    sTxt := CONCAT(sTxt, LREAL_TO_FMTSTR(REAL_TO_LREAL(GVL_Param.rLevelLow), 1, TRUE));
    sTxt := CONCAT(sTxt, ' %)');
    fbLog.Warn(sTxt);
END_IF

// -- SPX level high (> rLevelHigh) --
tonCoolHigh(IN := bCoolHigh, PT := tCooldown);
IF tonCoolHigh.Q THEN bCoolHigh := FALSE; END_IF
rtLevelHigh(CLK := GVL_Process.bWarnLevelHigh);
IF rtLevelHigh.Q AND NOT bCoolHigh THEN
    bCoolHigh := TRUE;
    sTxt := 'SPX level high: ';
    sTxt := CONCAT(sTxt, LREAL_TO_FMTSTR(REAL_TO_LREAL(GVL_IO.rSPXLevel), 1, TRUE));
    sTxt := CONCAT(sTxt, ' % (limit ');
    sTxt := CONCAT(sTxt, LREAL_TO_FMTSTR(REAL_TO_LREAL(GVL_Param.rLevelHigh), 1, TRUE));
    sTxt := CONCAT(sTxt, ' %)');
    fbLog.Warn(sTxt);
END_IF

// -- SPX tank empty (< rLevelEmpty) - lockout (fault 51 logs the [X]) --
tonCoolEmpty(IN := bCoolEmpty, PT := tCooldown);
IF tonCoolEmpty.Q THEN bCoolEmpty := FALSE; END_IF
rtLevelEmpty(CLK := GVL_Process.bLevelEmpty);
IF rtLevelEmpty.Q AND NOT bCoolEmpty THEN
    bCoolEmpty := TRUE;
    sTxt := 'SPX tank EMPTY: ';
    sTxt := CONCAT(sTxt, LREAL_TO_FMTSTR(REAL_TO_LREAL(GVL_IO.rSPXLevel), 1, TRUE));
    sTxt := CONCAT(sTxt, ' % (< ');
    sTxt := CONCAT(sTxt, LREAL_TO_FMTSTR(REAL_TO_LREAL(GVL_Param.rLevelEmpty), 1, TRUE));
    sTxt := CONCAT(sTxt, ' %) - pump stopped, mother release blocked');
    fbLog.Warn(sTxt);
END_IF

// -- bad SPX spray pressure (set after a stroke; cleared at cycle start) --
// (if it fires on the OPENING stroke, the T4 average shown is still
//  from the previous cycle - only T3 is fresh at that moment)
rtBadSPX(CLK := GVL_Process.bWarnBadSPX);
IF rtBadSPX.Q THEN
    sTxt := 'Bad SPX pressure: avg T3 ';
    sTxt := CONCAT(sTxt, LREAL_TO_FMTSTR(REAL_TO_LREAL(GVL_Process.rSPXAvgT3), 2, TRUE));
    sTxt := CONCAT(sTxt, ' / T4 ');
    sTxt := CONCAT(sTxt, LREAL_TO_FMTSTR(REAL_TO_LREAL(GVL_Process.rSPXAvgT4), 2, TRUE));
    sTxt := CONCAT(sTxt, ' bar (target ');
    sTxt := CONCAT(sTxt, LREAL_TO_FMTSTR(REAL_TO_LREAL(GVL_Param.rSPXPressureTarget), 2, TRUE));
    sTxt := CONCAT(sTxt, ' +/- ');
    sTxt := CONCAT(sTxt, LREAL_TO_FMTSTR(REAL_TO_LREAL(GVL_Param.rSPXPressTol), 2, TRUE));
    sTxt := CONCAT(sTxt, ')');
    fbLog.Warn(sTxt);
END_IF

// -- circulation pressure mismatch (recomputed at each cycle end) --
rtCircPress(CLK := GVL_Process.bWarnCircPress);
IF rtCircPress.Q THEN
    sTxt := 'Adjust circulation pressure: spray avg ';
    sTxt := CONCAT(sTxt, LREAL_TO_FMTSTR(REAL_TO_LREAL(GVL_Process.rSPXAvg), 2, TRUE));
    sTxt := CONCAT(sTxt, ' vs circulation avg ');
    sTxt := CONCAT(sTxt, LREAL_TO_FMTSTR(REAL_TO_LREAL(GVL_Process.rSPXAvgCirc), 2, TRUE));
    sTxt := CONCAT(sTxt, ' bar (tol ');
    sTxt := CONCAT(sTxt, LREAL_TO_FMTSTR(REAL_TO_LREAL(GVL_Param.rCircPressTol), 2, TRUE));
    sTxt := CONCAT(sTxt, ')');
    fbLog.Warn(sTxt);
END_IF

//------------------------------------------------------------------
// 4) PARAMETER SCREEN EVENTS  (PRG_Params runs earlier this scan;
//    bMsgTrig is TRUE for exactly the Apply/Reset press scan)
//------------------------------------------------------------------
rtParamMsg(CLK := PRG_Params.bMsgTrig);
IF rtParamMsg.Q THEN
    IF NOT PRG_Params.bLastApplyOk THEN
        // 'Rejected: sequence not idle' / 'Rejected: values must be > 0'
        sTxt := CONCAT('Parameters: ', PRG_Params.sParamStatus);
        fbLog.Warn(sTxt);
    ELSIF PRG_Params.sChangeList <> '' THEN
        // only the params that actually changed, old->new
        // (list is built by PRG_Params, where old and new coexist)
        IF PRG_Params.bLastWasReset THEN
            sTxt := 'Parameters RESET to defaults: ';
        ELSE
            sTxt := 'Parameters applied: ';
        END_IF
        sTxt := CONCAT(sTxt, PRG_Params.sChangeList);
        fbLog.Warn(sTxt);          // WARN so it shows on the Warnings dashboard
        bSnapReq := TRUE;          // and refresh the full snapshot right after
    END_IF
    // accepted but nothing changed -> stay silent (no log spam)
END_IF

//------------------------------------------------------------------
// 4b) PARAMETER SNAPSHOT  (full current values in ONE machine-parsable
//     INFO line - the Grafana "Current parameters" panels read this.
//     Written at boot, after every accepted Apply/Reset, and every
//     tSnapBeat as a heartbeat. Keep the 'key=value' format stable:
//     the dashboard regexes depend on it!)
//------------------------------------------------------------------
tonSnapBeat(IN := NOT tonSnapBeat.Q, PT := tSnapBeat);   // self-retriggering
IF tonSnapBeat.Q THEN
    bSnapReq := TRUE;
END_IF

IF bSnapReq AND fbLog.bTimeValid THEN
    bSnapReq := FALSE;
    // (T2/T6 and T3/T4 are always written as pairs by PRG_Params,
    //  so logging T2 and T3 represents both members of each pair)
    sTxt := 'Params snapshot: T1=';
    sTxt := CONCAT(sTxt, LREAL_TO_FMTSTR(TIME_TO_LREAL(GVL_Param.tDewaterTime) / 1000.0, 1, TRUE));
    sTxt := CONCAT(sTxt, 's T2/T6=');
    sTxt := CONCAT(sTxt, LREAL_TO_FMTSTR(TIME_TO_LREAL(GVL_Param.tSPXMaxOpenTime) / 1000.0, 1, TRUE));
    sTxt := CONCAT(sTxt, 's T3/T4=');
    sTxt := CONCAT(sTxt, LREAL_TO_FMTSTR(TIME_TO_LREAL(GVL_Param.tSprayOpenTime) / 1000.0, 1, TRUE));
    sTxt := CONCAT(sTxt, 's T5=');
    sTxt := CONCAT(sTxt, LREAL_TO_FMTSTR(TIME_TO_LREAL(GVL_Param.tSPXDewaterTime) / 1000.0, 1, TRUE));
    sTxt := CONCAT(sTxt, 's SPX=');
    sTxt := CONCAT(sTxt, LREAL_TO_FMTSTR(REAL_TO_LREAL(GVL_Param.rSPXPressureTarget), 2, TRUE));
    sTxt := CONCAT(sTxt, 'bar Pump=');
    sTxt := CONCAT(sTxt, LREAL_TO_FMTSTR(REAL_TO_LREAL(GVL_Param.rPumpSpeedBase), 1, TRUE));
    sTxt := CONCAT(sTxt, 'Hz');
    fbLog.Info(sTxt);
END_IF

//------------------------------------------------------------------
// 5) run the logger (drains the queue to the file)
//------------------------------------------------------------------
fbLog();

END_PROGRAM

// ---- POUs/FB_EventLog.TcPOU
FUNCTION_BLOCK FB_EventLog
//==================================================================
// CENTRAL EVENT LOGGER
//   Info() / Warn() / Error()  -> tagged, timestamped line -> queue
//   FB body (call once per scan) -> drains the queue to the file
//
//   Line format (tag FIRST so the eye can scan the left column):
//     [.]  2026-07-08-14:03:21.457  AUTO armed by operator
//     [!]  2026-07-08-14:05:02.113  SPX level low: 18.4 % (limit 20.0 %)
//     [X]  2026-07-08-14:07:44.902  FAULT 20: SPX valve stuck ...
//        [.] = INFO    [!] = WARN    [X] = ERROR
//   grep-friendly:  grep '^\[X\]' machine_events_2026-07.log
//
//   MONTHLY ROTATION: the file name is built per write as
//     <sBaseName>_YYYY-MM.log      e.g. machine_events_2026-07.log
//   so a new month automatically starts a new file (old months are
//   kept - clean them up manually or via cron/scheduled task).
//   On every PLC boot AND on each month rollover a legend/separator
//   header line is written first.
//
//   File location comes from GVL_Param.sLogDir:
//     ''  -> target's TwinCAT boot folder (portable default:
//            Windows C:\TwinCAT\3.1\Boot\ , BSD/Linux /usr/local/etc/TwinCAT/3.1/Boot\)
//     any full directory otherwise (per-machine, persistent).
//
//   Philosophy: NEVER block the machine. File error -> line dropped,
//   counted in nFailCount. Queue full -> line dropped, counted in
//   nDropped. Watch the outputs online if the file stays empty.
//
//   NOTE: call Info/Warn/Error only from the SAME PLC task that calls
//   the FB body (no locking inside).
//==================================================================
VAR_INPUT
    sBaseName : STRING(60) := 'machine_events';   // -> <base>_YYYY-MM.log; dir = GVL_Param.sLogDir
END_VAR
VAR_OUTPUT
    bTimeValid : BOOL;            // local clock ready (gate one-shot boot messages on this)
    nLastErrId : UDINT;           // last ADS error id from open/write
    nFailCount : UINT;            // lines lost to file errors
    nDropped   : UINT;            // lines lost to queue overflow
    sLastPath  : STRING(255);     // last path handed to FB_FileOpen (1st thing to check on Linux)
END_VAR
VAR
    // ---- timestamp ----
    fbTime  : FB_LocalSystemTime := (bEnable := TRUE, dwCycle := 1);

    // ---- ring buffer ----
    aQueue  : ARRAY[0..cQLAST] OF STRING(255);
    nHead   : INT;                // next free slot
    nTail   : INT;                // oldest queued line
    nCount  : INT;                // lines currently queued

    // ---- file access (Tc2_System) ----
    fbOpen  : FB_FileOpen;
    fbWrite : FB_FileWrite;
    fbClose : FB_FileClose;
    hFile   : UINT;
    eStep   : (IDLE, OPEN_FILE, WRITE_HDR, WRITE_LINE, CLOSE_FILE);
    sLine   : STRING(255);        // line currently being written
    sHdr    : STRING(120);        // legend/separator header

    // ---- monthly file name ----
    sCurFile  : STRING(80);       // name for the current month
    sLastFile : STRING(80);       // last name actually opened (header trigger)
    sMon      : STRING(4);

    // ---- path building ----
    sFullPath : STRING(255);
    ePathMode : E_OpenPath;       // PATH_BOOTPATH (portable) or PATH_GENERIC (explicit dir)
    sSep      : STRING(1);
END_VAR
VAR CONSTANT
    cQSIZE : INT := 16;
    cQLAST : INT := 15;
END_VAR

// ---- time base (cyclic) ----
fbTime();
bTimeValid := fbTime.bValid;

// ---- drain queue: open (append) -> [header] -> write burst -> close ----
CASE eStep OF

    IDLE:
        IF nCount > 0 THEN
            sLine  := aQueue[nTail];
            nTail  := (nTail + 1) MOD cQSIZE;
            nCount := nCount - 1;
            eStep  := OPEN_FILE;
        END_IF

    OPEN_FILE:
        // ---- monthly file name: <base>_YYYY-MM.log ----
        IF fbTime.bValid THEN
            sMon := WORD_TO_STRING(fbTime.systemTime.wMonth);
            IF fbTime.systemTime.wMonth < 10 THEN
                sMon := CONCAT('0', sMon);
            END_IF
            sCurFile := CONCAT(sBaseName, '_');
            sCurFile := CONCAT(sCurFile, WORD_TO_STRING(fbTime.systemTime.wYear));
            sCurFile := CONCAT(sCurFile, '-');
            sCurFile := CONCAT(sCurFile, sMon);
            sCurFile := CONCAT(sCurFile, '.log');
        ELSE
            sCurFile := CONCAT(sBaseName, '.log');   // clock not up yet (rare)
        END_IF

        // ---- directory: GVL_Param.sLogDir ('' = portable boot folder) ----
        // Resolved on every attempt -> sLogDir changes take effect on
        // the next event, no restart needed.
        IF GVL_Param.sLogDir = '' THEN
            sFullPath := sCurFile;        // portable default: target's boot folder
            ePathMode := PATH_BOOTPATH;
        ELSE
            sFullPath := GVL_Param.sLogDir;
            // append a trailing separator matching the path style if missing
            sSep := RIGHT(sFullPath, 1);
            IF sSep <> '/' AND sSep <> '\' THEN
                IF FIND(sFullPath, '/') > 0 THEN
                    sFullPath := CONCAT(sFullPath, '/');   // Linux-style
                ELSE
                    sFullPath := CONCAT(sFullPath, '\');   // Windows-style
                END_IF
            END_IF
            sFullPath := CONCAT(sFullPath, sCurFile);
            ePathMode := PATH_GENERIC;
        END_IF
        sLastPath := sFullPath;

        fbOpen(sNetId    := '',
               sPathName := sFullPath,
               nMode     := FOPEN_MODEAPPEND OR FOPEN_MODETEXT,
               ePath     := ePathMode,
               tTimeout  := T#3S,
               bExecute  := TRUE);
        IF NOT fbOpen.bBusy THEN
            fbOpen(bExecute := FALSE);
            IF fbOpen.bError THEN
                nLastErrId := fbOpen.nErrId;
                nFailCount := nFailCount + 1;
                eStep := IDLE;            // drop this line - never block the machine
            ELSE
                hFile := fbOpen.hFile;
                IF sCurFile <> sLastFile THEN
                    sLastFile := sCurFile;   // first write after boot, or month rollover
                    eStep := WRITE_HDR;      // -> drop the legend/separator first
                ELSE
                    eStep := WRITE_LINE;
                END_IF
            END_IF
        END_IF

    WRITE_HDR:
        sHdr := '==== log opened (PLC boot / month rollover) | legend: [.]=INFO  [!]=WARN  [X]=ERROR ====$N';
        fbWrite(sNetId     := '',
                hFile      := hFile,
                pWriteBuff := ADR(sHdr),
                cbWriteLen := TO_UDINT(LEN(sHdr)),
                tTimeout   := T#3S,
                bExecute   := TRUE);
        IF NOT fbWrite.bBusy THEN
            fbWrite(bExecute := FALSE);
            IF fbWrite.bError THEN
                nLastErrId := fbWrite.nErrId;
                nFailCount := nFailCount + 1;
            END_IF
            eStep := WRITE_LINE;          // header failure never blocks the real line
        END_IF

    WRITE_LINE:
        fbWrite(sNetId     := '',
                hFile      := hFile,
                pWriteBuff := ADR(sLine),
                cbWriteLen := TO_UDINT(LEN(sLine)),
                tTimeout   := T#3S,
                bExecute   := TRUE);
        IF NOT fbWrite.bBusy THEN
            fbWrite(bExecute := FALSE);
            IF fbWrite.bError THEN
                nLastErrId := fbWrite.nErrId;
                nFailCount := nFailCount + 1;
                eStep := CLOSE_FILE;      // always close after an error
            ELSIF nCount > 0 THEN
                // burst: everything queued goes out in ONE open/close session
                sLine  := aQueue[nTail];
                nTail  := (nTail + 1) MOD cQSIZE;
                nCount := nCount - 1;     // stay in WRITE_LINE -> re-triggers next scan
            ELSE
                eStep := CLOSE_FILE;
            END_IF
        END_IF

    CLOSE_FILE:
        fbClose(sNetId   := '',
                hFile    := hFile,
                tTimeout := T#3S,
                bExecute := TRUE);
        IF NOT fbClose.bBusy THEN
            fbClose(bExecute := FALSE);
            hFile := 0;
            eStep := IDLE;
        END_IF

END_CASE

METHOD Error : BOOL
VAR_INPUT
    sMsg : STRING(255);
END_VAR
Error := Push('[X]  ', sMsg);
END_METHOD

// INFO [.] = normal life of the machine (boot, mode, cycles, params, manual).
METHOD Info : BOOL   // TRUE = queued, FALSE = dropped (queue full)
VAR_INPUT
    sMsg : STRING(255);
END_VAR
Info := Push('[.]  ', sMsg);
END_METHOD

METHOD PRIVATE Push : BOOL
VAR_INPUT
    sTag : STRING(5);
    sMsg : STRING(255);
END_VAR
VAR
    sLn : STRING(255);
END_VAR
sLn := sTag;
// timestamp (placeholder during the first scans, before the clock is up)
IF fbTime.bValid THEN
    sLn := CONCAT(sLn, SYSTEMTIME_TO_STRING(fbTime.systemTime));
ELSE
    sLn := CONCAT(sLn, '????-??-??-??:??:??.???');
END_IF
sLn := CONCAT(sLn, '  ');
sLn := CONCAT(sLn, sMsg);
sLn := CONCAT(sLn, '$N');          // CONCAT truncates safely at 255 chars

IF nCount < cQSIZE THEN
    aQueue[nHead] := sLn;
    nHead  := (nHead + 1) MOD cQSIZE;
    nCount := nCount + 1;
    Push   := TRUE;
ELSE
    nDropped := nDropped + 1;      // queue full - drop, never block
    Push     := FALSE;
END_IF
END_METHOD

// WARN [!] = process warnings & rejected operations (machine keeps running).
METHOD Warn : BOOL   // TRUE = queued, FALSE = dropped (queue full)
VAR_INPUT
    sMsg : STRING(255);
END_VAR
Warn := Push('[!]  ', sMsg);
END_METHOD

END_FUNCTION_BLOCK

// ---- POUs/PRG_Telegram.TcPOU
PROGRAM PRG_Telegram
//==================================================================
// TELEGRAM FAULT NOTIFIER   (TF6760 / Tc3_IotBase)
//   Sends one message to a Telegram chat on every fault entry
//   (rising edge of MAIN.bError). Fire-and-forget: a failed send is
//   counted and dropped - the machine is never blocked.
//
//   Must be called AFTER PRG_Spray() in MAIN, so that
//   PRG_Spray.sErrorText is already updated on the fault scan.
//
//   Setup:
//     1. Telegram @BotFather -> /newbot -> paste the token into
//        GVL_Secrets.TELEGRAM_BOT_TOKEN (file is git-ignored).
//     2. Send any message to the bot, then open in a browser:
//          https://api.telegram.org/bot<TOKEN>/getUpdates
//        and copy  "chat":{"id":...}  into GVL_Secrets.TELEGRAM_CHAT_ID.
//        (For a group: add the bot to the group; the id is negative.)
//     3. License TF6760 on the target (7-day trial works for tests).
//     4. The target needs internet + DNS (ping api.telegram.org).
//==================================================================
VAR
    // ---- config (built on first scan from GVL_Secrets) ----
    sUri      : STRING(255);                  // '/bot<TOKEN>/sendMessage'
    sChatId   : STRING(31);                   // negative for group chats
    tCooldown : TIME := T#30S;                // min. spacing between messages

    // ---- HTTP client / request (Tc3_IotBase) ----
    fbClient  : FB_IotHttpClient := (sHostName := 'api.telegram.org',
                                     nHostPort := 443,
                                     bKeepAlive := FALSE);
    fbRequest : FB_IotHttpRequest;
    bTlsInit  : BOOL;                         // TLS + URI set before first Execute()

    // ---- event detection ----
    rtFault   : R_TRIG;                       // fault entry (MAIN.bError)
    tonCool   : TON;
    bCool     : BOOL;

    // ---- timestamp ----
    fbTime    : FB_LocalSystemTime := (bEnable := TRUE, dwCycle := 1);

    // ---- message buffers ----
    sText     : STRING(255);                  // human text (ASCII only!)
    sPending  : STRING(255);                  // one-slot queue (JSON body)
    sBody     : STRING(255);                  // JSON body currently sending
    eStep     : (IDLE, SEND, WAIT_RESPONSE);
    tonSendTo : TON;                          // give-up timer for SEND

    // ---- diagnostics (watch online if no message arrives) ----
    nLastStatus : UINT;                       // last HTTP status (200 = OK)
    nFailCount  : UINT;                       // messages lost to errors
END_VAR

//==================================================================
// First scan: build the URI from the (git-ignored) secrets GVL and
// configure TLS. Both must happen before the first Execute() call.
//==================================================================
IF NOT bTlsInit THEN
    bTlsInit := TRUE;

    sUri := CONCAT('/bot', GVL_Secrets.TELEGRAM_BOT_TOKEN);
    sUri := CONCAT(sUri, '/sendMessage');
    sChatId := GVL_Secrets.TELEGRAM_CHAT_ID;

    // Quick start: skip server-certificate verification.
    // For production, put a CA bundle (.pem) on the target and use:
    //   fbClient.stTLS.sCA := 'C:\TwinCAT\3.1\Boot\ca-bundle.pem';
    fbClient.stTLS.bNoServerCertCheck := TRUE;
END_IF

fbClient.Execute();      // background comms - MUST run every scan
fbTime();

//==================================================================
// Fault edge + cooldown  (same pattern as PRG_FileLogger)
//==================================================================
rtFault(CLK := MAIN.bError);

tonCool(IN := bCool, PT := tCooldown);
IF tonCool.Q THEN
    bCool := FALSE;
END_IF

IF rtFault.Q AND NOT bCool THEN
    bCool := TRUE;

